IF xDeleteProcessFlag_St1St2 THEN
	xDeleteProcessFlag_St1St2:=FALSE;
	TProcess.T_Ctrle.xAbordProcess:=FALSE;
	TProcess.T_Ctrle.xStop:=FALSE;
END_IF;
END_ACTION
ACTION CtrlFunctionButton:
(* Bt Function Button *)
	xTmp:=	NOT(xChangePage)
			AND T_Visu.T_CtrleAction.xDone
			AND NOT(T_Visu.T_CtrleAction.xExecute);
	IF (wForceMaskFunctionPanel <> 0) THEN
		(* Wurde von einer Funktion überschrieben *)
		T_ConfigPage.wMaskFunctionPanel:=wForceMaskFunctionPanel;
		T_ConfigPage.wMaskProcFunctionPanel:=wForceMaskFunctionPanel;
		wMaskFunctionPanel:=wForceMaskFunctionPanel;
		wForceMaskFunctionPanel:=0;
	END_IF;
	FOR ii:=1 TO 12 DO
		IF (aiForceRTrigActionFunctionPanel[ii] <> 0) THEN
			(* Wurde von einer Funktion überschrieben *)
			T_ConfigPage.aiRTrigActionFunctionPanel:=aiForceRTrigActionFunctionPanel;
			EXIT;
		END_IF;
	END_FOR;
	aiForceRTrigActionFunctionPanel:=aiDelectRTrigActionFunctionPanel;
	RisingEdgeBtFunctionPanel(CLK:=	(T_ExchgParam.T_BtFunctionPanel.wActivBt
									AND wMaskFunctionPanel) <> 16#0);
	IF xTmp THEN
		(* check if more than one button is pressed-->if only one Button than start the procedure *)
		IF xFct_CheckSingleButtonActivation(wInputButton:=T_ExchgParam.T_BtFunctionPanel.wActivBt) THEN
		(* activ action of rising edge *)
			IF RisingEdgeBtFunctionPanel.Q AND NOT(xTriggerWait) THEN
				ii:=iFct_GetBitNumber(wInputButton:=T_ExchgParam.T_BtFunctionPanel.wActivBt);
				IF (T_ConfigPage.aiRTrigActionFunctionPanel[ii] <> 0) THEN
					T_Visu.T_CtrleAction.iFunction:=T_ConfigPage.aiRTrigActionFunctionPanel[ii];
					T_Visu.T_CtrleAction.xExecute:=TRUE;
				END_IF;
			END_IF;
		END_IF;
	END_IF
END_ACTION
ACTION CtrlPanelLeftButton:
(* Bt Panel left *)
	xTmp:=	NOT(xChangePage)
			AND T_Visu.T_CtrleAction.xDone
			AND NOT(T_Visu.T_CtrleAction.xExecute)
			AND NOT(T_StartUp.T_State.xBlockChangeMovementVisu)
			AND NOT(T_Visu.T_CtrleAction.xFunctionActive)
			AND (T_ExchgParam.T_Visu.T_Message.iState <> 401)
			AND ((T_ExchgParam.T_Visu.bMachineState AND 16#2) <> 16#2);
	xParameterButtonBlocked:=NOT(xTmp);
	RisingEdgeBtPanelLeft(CLK:=		(wActivBtLeft
									AND wMaskBtPanelLeft) <> 16#0);

	FallingEdgeBtPanelLeft(CLK:=		(wActivBtLeft
									AND wMaskBtPanelLeft) <> 16#0);
	IF RisingEdgeBtPanelLeft.Q THEN
		wActivBtPanelLeft:=wActivBtLeft;
	END_IF;
	IF xTmp THEN
		(* check if more than one button is pressed-->if only one Button than start the procedure *)
		IF xFct_CheckSingleButtonActivation(wInputButton:=wActivBtPanelLeft) THEN
		(* activ action of rising edge *)
			IF RisingEdgeBtPanelLeft.Q THEN
				ii:=iFct_GetBitNumber(wInputButton:=wActivBtPanelLeft);
				IF (T_ConfigPage.aiRTrigActionPanelLeft[ii] <> 0) THEN
					T_Visu.T_CtrleAction.iFunction:=T_ConfigPage.aiRTrigActionPanelLeft[ii];
					T_Visu.T_CtrleAction.xExecute:=TRUE;
				END_IF;
			END_IF;
		END_IF;
	END_IF

(* Aktivierungsanzeige für Maschinen Lampe *)
	IF TMachineLamp.T_CtrleCyl.T_Standard.xActivOn THEN
		T_ExchgParam.T_TouchScreenBtPanel.iStateSetupLamp:=1;
	ELSE
		T_ExchgParam.T_TouchScreenBtPanel.iStateSetupLamp:=0;
	END_IF;

(* Auswahl der Seiten über die Recht Sondertasten *)
T_ExchgParam.T_TouchScreenBtPanel.iStateButtonPage:=0;
CASE T_Visu.T_PlcParam.dwActualPage OF
(* NormalMode	Task 1 *)
gT_PageNumber.iAutoMode_Process:				T_ExchgParam.T_TouchScreenBtPanel.iStateButtonPage:=16#20;
gT_PageNumber.iAutoMode_ProcessValue1:			T_ExchgParam.T_TouchScreenBtPanel.iStateButtonPage:=16#40;		(* IGS *)
gT_PageNumber.iAutoMode_ProcessValue2:			T_ExchgParam.T_TouchScreenBtPanel.iStateButtonPage:=16#80;		(* IGS *)
gT_PageNumber.iAutoMode_PartQuality:				T_ExchgParam.T_TouchScreenBtPanel.iStateButtonPage:=16#100;		(* alt 80 *)
(* NormalMode	Task 4 *)
gT_PageNumber.iAutoMode_ToolChange:			T_ExchgParam.T_TouchScreenBtPanel.iStateButtonPage:=16#20;
gT_PageNumber.iAutoMode_UserLevel:				T_ExchgParam.T_TouchScreenBtPanel.iStateButtonPage:=16#40;
gT_PageNumber.iAutoMode_Language:				T_ExchgParam.T_TouchScreenBtPanel.iStateButtonPage:=16#80;
(* NormalMode	Task 5 *)
gT_PageNumber.iAutoMode_WPCounter:				T_ExchgParam.T_TouchScreenBtPanel.iStateButtonPage:=16#20;
gT_PageNumber.iAutoMode_LampTest:				T_ExchgParam.T_TouchScreenBtPanel.iStateButtonPage:=16#40;
gT_PageNumber.iAutoMode_SafetyCheck:			T_ExchgParam.T_TouchScreenBtPanel.iStateButtonPage:=16#80;
gT_PageNumber.iAutoMode_SysInfo:				T_ExchgParam.T_TouchScreenBtPanel.iStateButtonPage:=16#100;

(* SetupMode A	Task 1 *)
gT_PageNumber.iHandMode_Process:				T_ExchgParam.T_TouchScreenBtPanel.iStateButtonPage:=16#20;
gT_PageNumber.iHandMode_WorkParameter:		T_ExchgParam.T_TouchScreenBtPanel.iStateButtonPage:=16#40;
gT_PageNumber.iHandMode_RegulatorPara:			T_ExchgParam.T_TouchScreenBtPanel.iStateButtonPage:=16#80;
gT_PageNumber.iHandMode_OnlineChange:			T_ExchgParam.T_TouchScreenBtPanel.iStateButtonPage:=16#100;	(* alt 40 *)
gT_PageNumber.iHandMode_ConfigPosition:			T_ExchgParam.T_TouchScreenBtPanel.iStateButtonPage:=16#200;	(* alt 80 *)

(* SetupMode B	Task 5 *)
gT_PageNumber.iWorkStation_Setup1:				T_ExchgParam.T_TouchScreenBtPanel.iStateButtonPage:=16#20;
gT_PageNumber.iWorkStation_Setup2:				T_ExchgParam.T_TouchScreenBtPanel.iStateButtonPage:=16#40;
gT_PageNumber.iWorkStation_Setup3:				T_ExchgParam.T_TouchScreenBtPanel.iStateButtonPage:=16#80;
gT_PageNumber.iWorkStation_Setup4:				T_ExchgParam.T_TouchScreenBtPanel.iStateButtonPage:=16#100;
gT_PageNumber.iWorkStation_Setup5:				T_ExchgParam.T_TouchScreenBtPanel.iStateButtonPage:=16#200;
END_CASE;
END_ACTION
ACTION CtrlPanelRightButton:
(* Bt Panel right *)
	xTmp:=	NOT(xChangePage)
			AND T_Visu.T_CtrleAction.xDone
			AND NOT(T_Visu.T_CtrleAction.xExecute);
	IF (wForceMaskBtPanelRight <> 0) THEN
		(* Wurde von einer Funktion überschrieben *)
		T_ConfigPage.wMaskBtPanelRight:=wForceMaskBtPanelRight;
		T_ConfigPage.wMaskProcBtPanelRight:=wForceMaskBtPanelRight;
		wMaskBtPanelRight:=wForceMaskBtPanelRight;
		wForceMaskBtPanelRight:=0;
	END_IF;
	FOR ii:=1 TO 5 DO
		IF (aiForceRTrigActionPanelRight[ii] <> 0) THEN
			(* Wurde von einer Funktion überschrieben *)
			T_ConfigPage.aiRTrigActionPanelRight:=aiForceRTrigActionPanelRight;
			EXIT;
		END_IF;
	END_FOR;
	aiForceRTrigActionPanelRight:=aiDeleteRTrigActionPanelRight;

	xActive_Joystick:=			IxJoystick_X_Plus OR IxJoystick_X_Minus OR IxJoystick_Y_Plus OR IxJoystick_Y_Minus;
	xActive_EnableSwitch:=		IxEnablingSwitchPlusButton OR IxEnablingSwitchMinusButton;

	IF (wActivBtRight = 0) AND NOT(xActive_EnableSwitch) THEN
		(* Achsenbewegung mit dem Joystick *)
		IF IxJoystick_Y_Plus AND NOT(IxJoystick_Y_Minus) AND gxEnable_Joystick_Axis_Z THEN
			wActivBtRight:=16#40;
			T_ConfigPage.aiRTrigActionPanelRight[2]:=216;
			wMaskBtPanelRight:=wActivBtRight;
		END_IF;
		IF NOT(IxJoystick_Y_Plus) AND IxJoystick_Y_Minus AND gxEnable_Joystick_Axis_Z THEN
			wActivBtRight:=16#20;
			T_ConfigPage.aiRTrigActionPanelRight[1]:=217;
			wMaskBtPanelRight:=wActivBtRight;
		END_IF;
		IF (IxJoystick_Y_Plus OR IxJoystick_Y_Minus) AND NOT(gxEnable_Joystick_Axis_Z) AND (T_ExchgParam.T_Visu.T_Message.iState <> 401) THEN
			T_ExchgParam.T_Visu.T_Message.iState:=306;	(* Warnung: Z Achse darf auf dieser Seite nicht verfahren werden ! *)
		END_IF;
	END_IF;

	IF (T_Visu.T_PlcParam.dwActualPage = gT_PageNumber.iWorkStation_Axis1) THEN
		gxReleaseEnableSwitch:=TRUE;
	ELSE
		gxReleaseEnableSwitch:=FALSE;
	END_IF;

	IF gxReleaseEnableSwitch AND (wActivBtRight = 0) AND NOT(xActive_Joystick) AND gT_SafetyStatus.xSecurityDoorOpen THEN
		(* Achsenbewegung mit dem Zustimmschalter *)
		IF IxEnablingSwitchPlusButton AND NOT(IxEnablingSwitchMinusButton) THEN
			wActivBtRight:=16#40;
			T_ConfigPage.aiRTrigActionPanelRight[2]:=216;
		END_IF;
		IF NOT(IxEnablingSwitchPlusButton) AND IxEnablingSwitchMinusButton THEN
			wActivBtRight:=16#20;
			T_ConfigPage.aiRTrigActionPanelRight[1]:=217;
		END_IF;
	END_IF;

	RisingEdgeBtPanelRight(CLK:=		(wActivBtRight
									AND wMaskBtPanelRight) <> 16#0);
	FallingEdgeBtPanelRight(CLK:=		(wActivBtRight
									AND wMaskBtPanelRight) <> 16#0);
	IF xTmp THEN
		(* check if more than one button is pressed-->if only one Button than start the procedure *)
		IF xFct_CheckSingleButtonActivation(wInputButton:=wActivBtRight) THEN
		(* activ action of rising edge *)
			IF RisingEdgeBtPanelRight.Q THEN
				ii:=iFct_GetBitNumber(wInputButton:=wActivBtRight) - 5;
				wActivBtPanelRight:=INT_TO_WORD(ii);
				IF (T_ConfigPage.aiRTrigActionPanelRight[ii] <> 0) THEN
					T_Visu.T_CtrleAction.iFunction:=T_ConfigPage.aiRTrigActionPanelRight[ii];
					T_Visu.T_CtrleAction.xExecute:=TRUE;
					xJogModeActive:=xFct_GetJogMode(iFunction:=T_Visu.T_CtrleAction.iFunction);
					wSaveBtPanelRight:=wActivBtRight;
				END_IF;
			END_IF;
		END_IF;
		(* activ action of failling edge *)
		IF FallingEdgeBtPanelRight.Q THEN
			ii:=WORD_TO_INT(wActivBtPanelRight);
			IF (T_ConfigPage.aiFTrigActionPanelRight[ii] <> 0) THEN
				T_Visu.T_CtrleAction.iFunction:=T_ConfigPage.aiFTrigActionPanelRight[ii];
				T_Visu.T_CtrleAction.xExecute:=TRUE;
			END_IF;
		END_IF;
	END_IF

(* Überprüfe wenn Jog Betrieb gestartet ist, dass wenn die Taste nicht mehr gedrückt ist, dass die Achse auch gestoppt wird-->Falls nicht, dann muss es explizit gestoppt werden *)
	IF xJogModeActive OR xTmpJogModeActive THEN
		CASE iStepJogModeActive OF
		1:	IF NOT(xInitJogVelocity) THEN
				xInitJogVelocity:=TRUE;
				lrJogVelocity:=T_ExchgParam.T_TeachIn.arTeachSelVel[ptrTCommonAxisActive^.T_Config_Gen.iTyp];
			END_IF;
			xJogModeActive:=FALSE;
			xTmpJogModeActive:=TRUE;
			IF ((wSaveBtPanelRight AND wActivBtRight) = 16#0) THEN
				(* Taste wurde losgelassen *)
				iStepJogModeActive:=iStepJogModeActive + 1;
				RETURN;
			END_IF;
			IF T_ExchgParam.T_TeachIn.xJogInc_Common_Setup_Axis AND (lrJogVelocity <> T_ExchgParam.T_TeachIn.arTeachSelVel[ptrTCommonAxisActive^.T_Config_Gen.iTyp]) THEN
				lrJogVelocity:=T_ExchgParam.T_TeachIn.arTeachSelVel[ptrTCommonAxisActive^.T_Config_Gen.iTyp];
				(* Jog-Betrieb ist ausgewählt-->Geschwindigkeit in Abhängigkeit des Poti einstellen *)
				IF NOT(ptrTCommonAxisActive^.T_CtrleSingle.xExecute) AND ptrTCommonAxisActive^.T_CtrleSingle.xDone AND
				     NOT(ptrTCommonAxisActive^.T_CtrleSingle.xErr) AND NOT(ptrTCommonAxisActive^.T_CtrleSingle.xNotMoving) THEN
					ptrTCommonAxisActive^.T_CtrleSingle.iFunction:=12;
					gxSetSpeedInMovement:=TRUE;
					IF ptrTCommonAxisActive^.T_CtrleSingle.xMovingForward THEN
						ptrTCommonAxisActive^.T_CtrleSingle.lrVelocity:=T_ExchgParam.T_TeachIn.arTeachSelVel[ptrTCommonAxisActive^.T_Config_Gen.iTyp];
					ELSE
						ptrTCommonAxisActive^.T_CtrleSingle.lrVelocity:=T_ExchgParam.T_TeachIn.arTeachSelVel[ptrTCommonAxisActive^.T_Config_Gen.iTyp]*-1.0;
					END_IF;
					ptrTCommonAxisActive^.T_CtrleSingle.xExecute:=TRUE;
				END_IF;
			END_IF;
		2:	IF ((ptrTCommonAxisActive^.T_CtrleSingle.iFunction = 6) OR (ptrTCommonAxisActive^.T_CtrleSingle.iFunction = 12)) AND NOT(ptrTCommonAxisActive^.T_CtrleSingle.xNotMoving) AND NOT(xJogModeActive) THEN
				T_Visu.T_CtrleAction.iFunction:=202;	(* Stoppen aller Achse *)
				T_Visu.T_CtrleAction.xExecute:=TRUE;
				xTmpJogModeActive:=FALSE;
				iStepJogModeActive:=1;
			END_IF
			IF (ptrTCommonAxisActive^.T_CtrleSingle.iFunction <> 6) AND (ptrTCommonAxisActive^.T_CtrleSingle.iFunction <> 12) AND NOT(xJogModeActive) THEN
				(* Es wurde ein Inkrementfahrt ausgelöst und daher muss es nicht explizit gestoppt werden *)
				xTmpJogModeActive:=FALSE;
				iStepJogModeActive:=1;
			END_IF;
			IF xJogModeActive THEN
				iStepJogModeActive:=1;	(* Jog wurde vor dem beenden wieder gestartet, daher muss es wieder überprüft werden *)
				xInitJogVelocity:=FALSE;
			END_IF;
		END_CASE;
	ELSE
		iStepJogModeActive:=1;
		xInitJogVelocity:=FALSE;
	END_IF;

(* Verwaltung der Freigabe für den Joystick *)
	IF NOT(T_StartUp.T_State.xCompleted) THEN
		(* Solange die Maschine nicht aufgestartet ist, ist die manuelle Achsenbewegung nicht erlaubt *)
		xResetEnableJoystickAxisZ:=TRUE;
		xSetEnableJoystickAxisZ:=FALSE;
	ELSIF NOT(gT_SafetyStatus.xSetupOperateModeActive) THEN
		(* Im NormalBetrieb ist die manuelle Achsenbewegung nicht erlaubt *)
		xResetEnableJoystickAxisZ:=TRUE;
		xSetEnableJoystickAxisZ:=FALSE;
	ELSIF gT_SafetyStatus.xSetupOperateModeActive AND (gT_SafetyStatus.iSetupMode = 1) THEN
		(* Im EinrichtBetrieb A ist die manuelle Achsenbewegung nur unter dem Task HandBetrieb erlaubt *)
		xResetEnableJoystickAxisZ:=TRUE;
		xSetEnableJoystickAxisZ:=FALSE;
		IF TStation_Work_St1.TControl.xEnable AND TStation_Work_St1.TControl.xRdy AND TStation_Work_St1.TControl.xDone AND NOT(TStation_Work_St1.TControl.xError) THEN
			IF (T_Visu.T_PlcParam.dwActualPage = gT_PageNumber.iHandMode_Process)
			OR (T_Visu.T_PlcParam.dwActualPage = gT_PageNumber.iHandMode_WorkParameter) OR (T_Visu.T_PlcParam.dwActualPage = gT_PageNumber.iHandMode_RegulatorPara)
			OR (T_Visu.T_PlcParam.dwActualPage = gT_PageNumber.iHandMode_OnlineChange) OR (T_Visu.T_PlcParam.dwActualPage = gT_PageNumber.iHandMode_ConfigPosition) THEN
				xResetEnableJoystickAxisZ:=FALSE;
				xSetEnableJoystickAxisZ:=TRUE;
			END_IF;
		END_IF;
	ELSIF gT_SafetyStatus.xSetupOperateModeActive AND (gT_SafetyStatus.iSetupMode = 2) THEN
		(* Im EinrichtBetrieb B ist die manuelle Achsenbewegung erlaubt sofern nicht eine Funktion am ausführen ist *)
		IF NOT(TStation_Work_St1.TControl.xEnable) OR NOT(TStation_Work_St1.TControl.xRdy) OR NOT(TStation_Work_St1.TControl.xDone) OR  TStation_Work_St1.TControl.xError THEN
			xResetEnableJoystickAxisZ:=TRUE;
			xSetEnableJoystickAxisZ:=FALSE;
		ELSE
			xResetEnableJoystickAxisZ:=FALSE;
			xSetEnableJoystickAxisZ:=TRUE;
		END_IF;
		IF xTmpStationSetupAxisZFunction AND (T_ExchgParam.T_StationCommon.iZAxisFirstSetup_ShowObjectNr = 3) THEN
			xResetEnableJoystickAxisZ:=FALSE;
			xSetEnableJoystickAxisZ:=TRUE;
		END_IF;
		IF xTmpStationSetupAxisZFunction AND (T_ExchgParam.T_StationCommon.iZAxisFirstSetup_ShowObjectNr <> 3) THEN
			xResetEnableJoystickAxisZ:=TRUE;
			xSetEnableJoystickAxisZ:=FALSE;
		END_IF;
		IF xTmpStationSetupAxisZFunctionToolGuide AND (T_ExchgParam.T_StationCommon.iZAxisGuideTube_ShowObjectNr = 6) THEN
			xResetEnableJoystickAxisZ:=FALSE;
			xSetEnableJoystickAxisZ:=TRUE;
		END_IF;
		IF xTmpStationSetupAxisZFunctionToolGuide AND (T_ExchgParam.T_StationCommon.iZAxisGuideTube_ShowObjectNr <> 6) THEN
			xResetEnableJoystickAxisZ:=TRUE;
			xSetEnableJoystickAxisZ:=FALSE;
		END_IF;
	ELSE
		(* Alles restliche ist nicht erlaubt *)
		xResetEnableJoystickAxisZ:=TRUE;
		xSetEnableJoystickAxisZ:=FALSE;
	END_IF;

	IF xSetEnableJoystickAxisZ THEN
		gxEnable_Joystick_Axis_Z:=TRUE;
	END_IF;
	IF xResetEnableJoystickAxisZ OR NOT(T_StartUp.T_Ctrle.xDone) THEN
		gxEnable_Joystick_Axis_Z:=FALSE;
	END_IF;
END_ACTION
ACTION CtrlParaListButton:
IF NOT(xSecurityKey) THEN
	iStationActive:=0;
ELSE
	iStationActive:=iSetupMode;
END_IF;
(* Bt Parameter List Button *)
	xTmp:=	NOT(xChangePage)
			AND T_Visu.T_CtrleAction.xDone
			AND NOT(T_Visu.T_CtrleAction.xExecute);
	RisingEdgeBtParameterList(CLK:=	(T_ExchgParam.T_BtParameterList.wActivBt<>0));
	IF xTmp THEN
		(* check if more than one button is pressed-->if only one Button than start the procedure *)
		IF xFct_CheckSingleButtonActivation(wInputButton:=T_ExchgParam.T_BtParameterList.wActivBt) THEN
		(* activ action of rising edge *)
			IF RisingEdgeBtParameterList.Q THEN
				ii:=iFct_GetBitNumber(wInputButton:=T_ExchgParam.T_BtParameterList.wActivBt);
				jj:=iFct_GetBitNumber(wInputButton:=awSaveStateTaskBar[iStationActive]);
(*				aiTempActiveParaListState[iStationActive,jj]:=ii;*)
				(* Da diese Software keine Parameterlisten bezogen auf Task hat, sind alle gleichgestellt *)
				aiTempActiveParaListState[iStationActive,1]:=ii;
				aiTempActiveParaListState[iStationActive,2]:=ii;
				aiTempActiveParaListState[iStationActive,3]:=ii;
				aiTempActiveParaListState[iStationActive,4]:=ii;
				aiTempActiveParaListState[iStationActive,5]:=ii;
				aiTempActiveParaListState[iStationActive,6]:=ii;
				xUpdateStationParameter:=TRUE;
			END_IF;
		END_IF;
		T_ExchgParam.T_BtParameterList.wActivBt:=0;
	ELSE
		T_ExchgParam.T_BtParameterList.wActivBt:=0;
	END_IF

FBGetParameterList(	xNormalModeActive:= NOT(xSecurityKey),
					iSetupMode:= iSetupMode,
					wActiveTaskBar:= awSaveStateTaskBar[iStationActive],
					aiTempActiveParaListState:= aiTempActiveParaListState,
					iActLevel:=T_ExchgParam.T_Visu.T_Level.iActLevel);
T_ExchgParam.T_BtParameterList.iEditParam:=FBGetParameterList.iParameterList;
T_ExchgParam.T_BtParameterList.wNotMasktext:=FBGetParameterList.wNotMasktext;
T_ExchgParam.T_BtParameterList.wState:=FBGetParameterList.wState;
T_ExchgParam.T_BtParameterList.aiSelectText:=FBGetParameterList.aiSelectText;
T_ExchgParam.T_BtParameterList.bParameterListEditable:=FBGetParameterList.bParameterListEditable;
T_ExchgParam.T_BtParameterList.bMessageParameter:=FBGetParameterList.bMessageParameter;
END_ACTION
ACTION CtrlPreWarning:
(* Ausgabe der Vorwarnungsmeldungen *)
IF T_ExchgParam.T_SafetyCtrl.xReadNextPreWarningMessage THEN
	T_ExchgParam.T_SafetyCtrl.xReadNextPreWarningMessage:=FALSE;
	IF gT_PreWarning.xPreWarningActive THEN
		iMessageSelected:=iMessageSelected + 1;
		IF (iMessageSelected > gT_PreWarning.iNumberOfMessage) THEN
			iMessageSelected:=gT_PreWarning.iNumberOfMessage;
		END_IF;
	END_IF;
END_IF;
IF T_ExchgParam.T_SafetyCtrl.xReadPreviousPreWarningMessage THEN
	T_ExchgParam.T_SafetyCtrl.xReadPreviousPreWarningMessage:=FALSE;
	IF gT_PreWarning.xPreWarningActive THEN
		iMessageSelected:=iMessageSelected - 1;
		IF (iMessageSelected < 1) THEN
			iMessageSelected:=1;
		END_IF;
	END_IF;
END_IF;
IF (iMessageSelected > gT_PreWarning.iNumberOfMessage) THEN
	iMessageSelected:=gT_PreWarning.iNumberOfMessage;
END_IF;
IF (iMessageSelected = 0) AND (gT_PreWarning.iNumberOfMessage > 0) THEN
	iMessageSelected:=1;
END_IF;
IF NOT(gT_PreWarning.xPreWarningActive) THEN
	T_ExchgParam.T_SafetyCtrl.sDynMsgPreWarningLine1Engl:=gT_PreWarning.asEmptyMessageEngl[1];
	T_ExchgParam.T_SafetyCtrl.sDynMsgPreWarningLine2Engl:=gT_PreWarning.asEmptyMessageEngl[2];
	T_ExchgParam.T_SafetyCtrl.sDynMsgPreWarningLine3Engl:=gT_PreWarning.asEmptyMessageEngl[3];
	T_ExchgParam.T_SafetyCtrl.sDynMsgPreWarningLine4Engl:=gT_PreWarning.asEmptyMessageEngl[4];
	T_ExchgParam.T_SafetyCtrl.sDynMsgPreWarningLine5Engl:=gT_PreWarning.asEmptyMessageEngl[5];
	T_ExchgParam.T_SafetyCtrl.sDynMsgPreWarningLine1Ger:=gT_PreWarning.asEmptyMessageGer[1];
	T_ExchgParam.T_SafetyCtrl.sDynMsgPreWarningLine2Ger:=gT_PreWarning.asEmptyMessageGer[2];
	T_ExchgParam.T_SafetyCtrl.sDynMsgPreWarningLine3Ger:=gT_PreWarning.asEmptyMessageGer[3];
	T_ExchgParam.T_SafetyCtrl.sDynMsgPreWarningLine4Ger:=gT_PreWarning.asEmptyMessageGer[4];
	T_ExchgParam.T_SafetyCtrl.sDynMsgPreWarningLine5Ger:=gT_PreWarning.asEmptyMessageGer[5];
ELSE
	sWrapTextEngl:='Message ';
	sWrapTextEngl:=CONCAT(sWrapTextEngl, INT_TO_STRING(iMessageSelected));
	sWrapTextEngl:=CONCAT(sWrapTextEngl, ' of ');
	sWrapTextEngl:=CONCAT(sWrapTextEngl, INT_TO_STRING(gT_PreWarning.iNumberOfMessage));
	T_ExchgParam.T_SafetyCtrl.sDynMsgPreWarningLine1Engl:=sWrapTextEngl;
	T_ExchgParam.T_SafetyCtrl.sDynMsgPreWarningLine2Engl:=gT_PreWarning.asMessageBufferEngl[iMessageSelected,2];
	T_ExchgParam.T_SafetyCtrl.sDynMsgPreWarningLine3Engl:=gT_PreWarning.asMessageBufferEngl[iMessageSelected,3];
	T_ExchgParam.T_SafetyCtrl.sDynMsgPreWarningLine4Engl:=gT_PreWarning.asMessageBufferEngl[iMessageSelected,4];
	T_ExchgParam.T_SafetyCtrl.sDynMsgPreWarningLine5Engl:=gT_PreWarning.asMessageBufferEngl[iMessageSelected,5];
	sWrapTextGer:='Meldung ';
	sWrapTextGer:=CONCAT(sWrapTextGer, INT_TO_STRING(iMessageSelected));
	sWrapTextGer:=CONCAT(sWrapTextGer, ' von ');
	sWrapTextGer:=CONCAT(sWrapTextGer, INT_TO_STRING(gT_PreWarning.iNumberOfMessage));
	T_ExchgParam.T_SafetyCtrl.sDynMsgPreWarningLine1Ger:=sWrapTextGer;
	T_ExchgParam.T_SafetyCtrl.sDynMsgPreWarningLine2Ger:=gT_PreWarning.asMessageBufferGer[iMessageSelected,2];
	T_ExchgParam.T_SafetyCtrl.sDynMsgPreWarningLine3Ger:=gT_PreWarning.asMessageBufferGer[iMessageSelected,3];
	T_ExchgParam.T_SafetyCtrl.sDynMsgPreWarningLine4Ger:=gT_PreWarning.asMessageBufferGer[iMessageSelected,4];
	T_ExchgParam.T_SafetyCtrl.sDynMsgPreWarningLine5Ger:=gT_PreWarning.asMessageBufferGer[iMessageSelected,5];
END_IF;
IF T_ExchgParam.T_SafetyCtrl.xResetMsgPreWarning THEN
	T_ExchgParam.T_SafetyCtrl.xResetMsgPreWarning:=FALSE;
	IF gT_PreWarning.xPreWarningActive AND (iMessageSelected <> 0) THEN
		giDeleteMessageNumber:=giDeleteMessageNumber + 1;
		gT_PreWarning.aiDeleteMessage[giDeleteMessageNumber]:=gT_PreWarning.aiMessageNrBuffer[iMessageSelected];
	END_IF;
END_IF;
IF T_ExchgParam.T_SafetyCtrl.xConfirmMsgPreWarning THEN
	T_ExchgParam.T_SafetyCtrl.xConfirmMsgPreWarning:=FALSE;
	T_ExchgParam.T_SafetyCtrl.bStateMessagePreWarning:=0;
END_IF;
IF (T_ExchgParam.T_SafetyCtrl.bStateMessageError <> 0) OR (T_ExchgParam.T_SafetyCtrl.bStateMessageInfo <> 0) OR (T_ExchgParam.T_SafetyCtrl.bStateMessageWarning <> 0) THEN
	T_ExchgParam.T_SafetyCtrl.xConfirmMsgPreWarning:=FALSE;
	T_ExchgParam.T_SafetyCtrl.bStateMessagePreWarning:=0;
END_IF;
END_ACTION
ACTION CtrlProcessFunction:
(* Manage process execution *)
	(* ...done *)
	RisingEdgeProcessDone(CLK:=T_Visu.T_CtrleProcess.xDone);
	IF RisingEdgeProcessDone.Q THEN
		;
	END_IF
	(* ...error *)
	RisingEdgeProcessError(CLK:=T_Visu.T_CtrleProcess.xErr);
	IF RisingEdgeProcessError.Q THEN
		(* Init. variable *)
		T_Visu.T_CtrleProcess.xExecute:=FALSE;
		T_Visu.T_CtrleProcess.xDone:=TRUE;
		T_Visu.T_CtrleProcess.xErr:=FALSE;
		T_Visu.T_CtrleProcess.udiErrorID:=0;
		iStepProcess:=1;
		xStepProcessDone:=FALSE;
	END_IF
	(* ...reset *)
	RisingEdgeReseTProcess(CLK:=T_Visu.T_CtrleProcess.xReset);
	IF RisingEdgeReseTProcess.Q THEN
		(* Init. variable *)
		T_Visu.T_CtrleProcess.xExecute:=FALSE;
		T_Visu.T_CtrleProcess.xDone:=TRUE;
		T_Visu.T_CtrleProcess.xErr:=FALSE;
		T_Visu.T_CtrleProcess.udiErrorID:=0;
		iStepProcess:=1;
		xStepProcessDone:=FALSE;
		(* Release process *)
		T_Visu.T_CtrleProcess.xReset:=FALSE;
		xProcessMachine:=FALSE;
		xProcessStation:=FALSE;
	END_IF
	RisingEdgeExecuteProcess(CLK:=T_Visu.T_CtrleProcess.xExecute);
	IF RisingEdgeExecuteProcess.Q THEN
		(* Release execution *)
		T_Visu.T_CtrleProcess.xExecute:=FALSE;
		CASE T_Visu.T_CtrleProcess.iFunction OF
		(* Process machine *)
		1:	xProcessMachine:=TRUE;
		(* Process station mit WstkTeller *)
		2:	xProcessStation:=TRUE;
		(* process not implemented *)
		ELSE	T_Visu.T_CtrleProcess.xDone:=FALSE;
				T_Visu.T_CtrleProcess.xErr:=TRUE;
				T_Visu.T_CtrleProcess.udiErrorID:=16#E000;
				(* exit FB *)
				RETURN;
		END_CASE
		(* Init. variable *)
		T_Visu.T_CtrleProcess.xDone:=FALSE;
		T_Visu.T_CtrleProcess.xErr:=FALSE;
		T_Visu.T_CtrleProcess.udiErrorID:=0;
		iStepProcess:=1;
		xStepProcessDone:=FALSE;
		(* exit FB *)
		RETURN;
	END_IF

(* Prozesse die im Einrichtbetrieb ausgelöst werden mit dem WstkTeller *)
	IF xProcessStation THEN
		IF NOT(TProcess.T_Ctrle.xExecute)  AND TProcess.T_Ctrle.xError AND TProcess.T_Ctrle.xErrorReady THEN
			iStepProcess:=90;
		END_IF;
		CASE iStepProcess OF
		1:	TProcess.T_Ctrle.xExecute:=TRUE;	(* Starten des Prozesses *)
			iStepProcess:=90;
		(* Abwarten auf das Prozessende *)
		90:	IF NOT(TProcess.T_Ctrle.xExecute)  AND (TProcess.T_Ctrle.xDone OR TProcess.T_Ctrle.xError) THEN
				T_StartUp.T_State.xBlockChangeMovementVisu:=FALSE;
				xProcessStation:=FALSE;
				T_Visu.T_CtrleProcess.xDone:=TRUE;
				T_Visu.T_CtrleProcess.xErr:=FALSE;
				T_Visu.T_CtrleProcess.udiErrorID:=0;
			END_IF;
			IF (T_ExchgParam.byOverride = 0) THEN
				T_ExchgParam.T_Visu.T_Message.iState:=330;	(* Override ist auf 0% gesetzt-->Keine Achsenbewegung ! *)
			ELSE
				IF (T_ExchgParam.T_Visu.T_Message.iState = 330) THEN
					T_ExchgParam.T_Visu.T_Message.iState:=0;
				END_IF;
			END_IF;
		END_CASE;
	END_IF;

(* Prozesse die im Automat ausgelöst werden *)
	IF xProcessMachine THEN
		CASE iStepProcess OF
		(* Überprüfe zuerst den WzWechsel der Bearbeitungsstationen *)
		1:	xProcessEnded:=FALSE;
			IF (TProcess.T_Ctrle.iFunctNr = 2) THEN
				(* Gilt nur für den Automat *)
				T_ExchgParam.T_Visu.T_Message.iState:=0;
				T_ExchgParam.T_StationCommon.T_ToolCounter_St1.diToolCycleCounter:=T_NovRam.T_Parameter.T_StationWork[gciStationSt1].T_ToolCounter.diToolCycleCounter;
				T_ExchgParam.T_StationCommon.T_ToolCounter_St1.diMaxNumberToolCycle:=T_NovRam.T_Parameter.T_StationWork[gciStationSt1].T_ToolCounter.diMaxNumberToolCycle;
				xTmp:=	((T_NovRam.T_Parameter.T_StationWork[gciStationSt1].T_ToolCounter.diMaxNumberToolCycle <> 0) AND
						(T_NovRam.T_Parameter.T_StationWork[gciStationSt1].T_ToolCounter.diToolCycleCounter >= T_NovRam.T_Parameter.T_StationWork[gciStationSt1].T_ToolCounter.diMaxNumberToolCycle));
				IF xTmp THEN
					T_ExchgParam.T_SafetyCtrl.bStateMessageRequest:=1;
					T_ExchgParam.T_SafetyCtrl.bStateMessagePreWarning:=0;
					T_StartUp.T_State.xBlockChangeMovementVisu:=TRUE;
					iStepProcess:=iStepProcess + 1;
				ELSE
					iStepProcess:=4;	(* Überprüfen des Namen für die Prozessanalyse *)
				END_IF;
			ELSE
					iStepProcess:=19;	(* Prozess kann gestartet werden *)
			END_IF;
			xProcessAbordet:=FALSE;
		(* Aufforderung an Operator für Eingabe ob WzWechsel stattgefunden hat oder nicht *)
		2:	IF T_ExchgParam.T_SafetyCtrl.xConfirmMsgRequest THEN
				T_ExchgParam.T_SafetyCtrl.xConfirmMsgRequest:=FALSE;
				T_ExchgParam.T_SafetyCtrl.bStateMessageRequest:=0;
				IF (T_ExchgParam.T_SafetyCtrl.bState_Select_St1 = 1) THEN
					T_NovRam.T_Parameter.T_StationWork[gciStationSt1].T_ToolCounter.diToolCycleCounter:=0;
					T_ExchgParam.T_StationCommon.T_ToolCounter_St1.diToolCycleCounter:=0;
				END_IF;
				TONWaitReadyStartButton(IN:=FALSE);
				T_ExchgParam.T_Visu.T_Message.iState:=101;	(* Aufforderung: Bitte StartTaste drücken um Prozess zu starten *)
				iStepProcess:=iStepProcess + 1;
			END_IF;
		(* Auffordern erneut die StartTaste zu drücken *)
		3:	T_CtrleBtStartStop.xForceSetStartButton:=TONWaitReadyStartButton.Q;
			T_CtrleBtStartStop.xForceSetStopButton:=TONWaitReadyStartButton.Q;
			T_ExchgParam.T_Visu.T_Message.iState:=101;	(* Aufforderung: Bitte StartTaste drücken um Prozess zu starten *)
			IF xStartButton THEN
				TONWaitReadyStartButton(IN:=FALSE);
				T_ExchgParam.T_Visu.T_Message.iState:=0;		(* Meldung zurücksetzen *)
				T_StartUp.T_State.xBlockChangeMovementVisu:=FALSE;
				iStepProcess:=4;
			END_IF;
			IF xStopButton THEN
				TONWaitReadyStartButton(IN:=FALSE);
				T_ExchgParam.T_Visu.T_Message.iState:=0;		(* Meldung zurücksetzen *)
				T_ExchgParam.T_Visu.T_Message.iState:=0;
				xProcessMachine:=FALSE;
				T_Visu.T_CtrleProcess.xDone:=TRUE;
				T_Visu.T_CtrleProcess.xErr:=FALSE;
				T_Visu.T_CtrleProcess.udiErrorID:=0;
				T_StartUp.T_State.xBlockChangeMovementVisu:=FALSE;
			END_IF;
		(* Überprüfe ob der Name für die Prozessanalyse eingegeben werden muss *)
		4:	IF (T_NovRam.T_Parameter.T_PartAnalysis[gciStationSt1].sStartOfProcess = '') THEN
				TStation_Work_St1.THWWorkStation.TCtrlWork.xWP_Analyse_StartAutomat:=TRUE;			(* Gilt für die Aufzeichnungsdatei, um festzulegen wann der Automat für die jeweilige Datei gestartet wurde *)
			END_IF;
			iStepProcess:=19;
		(* Sicherheitstüren Zuhaltung aktivieren *)
		19:	T_ExchgParam.T_SafetyCtrl.xCloseSecurityDoorMachine:=TRUE;
			iStepProcess:=20;
		20:	IF NOT(T_ExchgParam.T_SafetyCtrl.xCloseSecurityDoorMachine) THEN
				iStepProcess:=30;
			END_IF;
		(* Prozess starten *)
		30:	TProcess.T_Ctrle.xExecute:=TRUE;	(* Starten des Prozesses *)
			iStepProcess:=90;
		90:	IF NOT(TProcess.T_Ctrle.xExecute)  AND TProcess.T_Ctrle.xDone THEN
				xProcessEnded:=TRUE;
				IF NOT(xProcessAbordet) THEN
					IF (TProcess.T_Ctrle.iFunctNr = 1) THEN
						T_StartUp.T_Ctrle.iMsgNumber:=3;	(* Die Maschine wurde Referenziert/Grundstellung! Bestätigen Sie die Meldung und die Zuhaltung der MaschinenTüre wird deaktiviert! *)
						T_StartUp.T_Ctrle.iFunction:=11;
						T_StartUp.T_Ctrle.xExecute:=TRUE;
					ELSIF (TProcess.T_Ctrle.iFunctNr = 2) THEN
						T_StartUp.T_Ctrle.iMsgNumber:=10;	(* Das Leerfahren im Automat ist beendet! Bestätigen Sie die Meldung und die Zuhaltung der MaschinenTüre wird deaktiviert! *)
						T_StartUp.T_Ctrle.iFunction:=11;
						T_StartUp.T_Ctrle.xExecute:=TRUE;
					END_IF;
				ELSE
					xProcessAbordet:=FALSE;
					T_StartUp.T_Ctrle.iMsgNumber:=10;	(* Prozess wurde abgebrochen! Bestätigen Sie die Meldung und die Zuhaltung der MaschinenTüre wird deaktiviert! *)
					T_StartUp.T_Ctrle.iFunction:=12;
					T_StartUp.T_Ctrle.xExecute:=TRUE;
				END_IF;
				T_StartUp.T_Ctrle.xUnlockSecurityDoor:=TRUE;	(* Auffordern Sicherheitstüren zu öffnen, nachdem die Meldung vom Operator Quittiert wurde *)
				xProcessMachine:=FALSE;
				T_Visu.T_CtrleProcess.xDone:=TRUE;
				T_Visu.T_CtrleProcess.xErr:=FALSE;
				T_Visu.T_CtrleProcess.udiErrorID:=0;
				T_ExchgParam.T_StationCommon.xBlockSelectAutoMode:=FALSE;
			END_IF;
			IF NOT(TProcess.T_Ctrle.xExecute)  AND TProcess.T_Ctrle.xError AND TProcess.T_Ctrle.xErrorReady THEN
				xProcessEnded:=TRUE;
				IF (TProcess.T_Ctrle.iFunctNr = 1) THEN
					T_StartUp.T_Ctrle.iMsgNumber:=58;	(* Während der Maschinen Ref./Grundstellung ist ein Fehler/Error aufgetreten! Bestätigen Sie die Meldung und Überprüfen Sie den entsprechenden Fehler/Error *)
				ELSIF (TProcess.T_Ctrle.iFunctNr = 2) THEN
					T_StartUp.T_Ctrle.iMsgNumber:=55;	(* Während des Automat ist ein Fehler/Error aufgetreten! Bestätigen Sie die Meldung und Überprüfen Sie den entsprechenden Fehler/Error *)
				END_IF;
				T_StartUp.T_Ctrle.iFunction:=10;
				T_StartUp.T_Ctrle.xUnlockSecurityDoor:=TRUE;	(* Auffordern Sicherheitstüren zu öffnen, nachdem die Meldung vom Operator Quittiert wurde *)
				T_StartUp.T_Ctrle.xExecute:=TRUE;
				xProcessMachine:=FALSE;
				T_Visu.T_CtrleProcess.xDone:=TRUE;
				T_Visu.T_CtrleProcess.xErr:=FALSE;
				T_Visu.T_CtrleProcess.udiErrorID:=0;
				T_ExchgParam.T_StationCommon.xBlockSelectAutoMode:=FALSE;
			END_IF;
			IF (T_ExchgParam.byOverride = 0) THEN
				T_ExchgParam.T_Visu.T_Message.iState:=330;	(* Override ist auf 0% gesetzt-->Keine Achsenbewegung ! *)
			ELSE
				IF (T_ExchgParam.T_Visu.T_Message.iState = 330) THEN
					T_ExchgParam.T_Visu.T_Message.iState:=0;
				END_IF;
			END_IF;
		END_CASE;
	END_IF;

	IF (T_StartUp.T_Ctrle.iMsgNumber = 10) AND (T_StartUp.T_Ctrle.iFunction = 11) AND NOT(T_StartUp.T_Ctrle.xDone) AND T_StartUp.T_State.xCompleted AND NOT(gT_SafetyStatus.xSetupOperateModeActive) AND NOT(T_ExchgParam.T_SafetyCtrl.xConfirmMsgInfo) THEN
		TONWaitSwitchOffMessage(IN:=TRUE,PT:=T#3s);
		IF TONWaitSwitchOffMessage.Q THEN
			T_ExchgParam.T_SafetyCtrl.xConfirmMsgInfo:=TRUE;
			TONWaitSwitchOffMessage(IN:=FALSE);
		END_IF;
	ELSE
		TONWaitSwitchOffMessage(IN:=FALSE);
	END_IF;

(* Ausgabe ob der Prozesszustand Aktiv ist *)
	T_ExchgParam.T_Visu.xActiveProcessState_St1St2:=	(T_NovRam.T_Parameter.T_PartAnalysis[gciStationSt1].sFileName <> '') OR (T_NovRam.T_Parameter.T_PartAnalysis[gciStationSt1].diActual_NumberHoleToWork <> 0);
	TProcess.T_Ctrle.xActiveProcessState:=T_ExchgParam.T_Visu.xActiveProcessState_St1St2;

(* Ausgabe der abgelaufenen Automat Prozesszeit *)
T_ExchgParam.T_StationCommon.T_Param_Machine.T_ParamAutomat.tAutoProcessTime_St1St2:=
										T_NovRam.T_Parameter.T_Machine.T_ParamAutomat.tAutoProcessTime_St1St2;
T_ExchgParam.T_StationCommon.T_Param_Machine.T_ParamAutomat.iAutoProcessDay_St1St2:=
										T_NovRam.T_Parameter.T_Machine.T_ParamAutomat.iAutoProcessDay_St1St2;

(* Ausgabe der Anzahl bearbeitenden Wstk *)
T_ExchgParam.T_StationCommon.T_Param_Machine.T_ParamAutomat.diNumberPartWorked_St1St2:=
										T_NovRam.T_Parameter.T_Machine.T_ParamAutomat.diNumberPartWorked_St1St2;

(* Eingabe WzWechsel *)
IF (T_ExchgParam.T_SafetyCtrl.bStateMessageRequest <> 0) THEN
	IF T_ExchgParam.T_SafetyCtrl.xSelect_ToolChange_St1 THEN
		T_ExchgParam.T_SafetyCtrl.xSelect_ToolChange_St1:=FALSE;
		IF (T_ExchgParam.T_SafetyCtrl.bState_Select_St1 = 0) THEN
			T_ExchgParam.T_SafetyCtrl.bState_Select_St1:=1;
		ELSIF (T_ExchgParam.T_SafetyCtrl.bState_Select_St1 = 1) THEN
			T_ExchgParam.T_SafetyCtrl.bState_Select_St1:=0;
		END_IF;
	END_IF;
ELSE
	T_ExchgParam.T_SafetyCtrl.bState_Select_St1:=0;
	T_ExchgParam.T_SafetyCtrl.xSelect_ToolChange_St1:=FALSE;
END_IF;

T_ExchgParam.T_StationCommon.T_Param_StationWork.T_TorqueSystem.rActual_Torque:=T_NovRam.T_Parameter.T_StationWork[1].T_TorqueSystem.rActual_Torque;
T_ExchgParam.T_StationCommon.T_Param_StationWork.T_TorqueSystem_L.rActual_Torque:=T_NovRam.T_Parameter.T_StationWork[1].T_TorqueSystem_L.rActual_Torque;
T_ExchgParam.T_StationCommon.T_Param_StationWork.T_TorqueSystem_M.rActual_Torque:=T_NovRam.T_Parameter.T_StationWork[1].T_TorqueSystem_M.rActual_Torque;
END_ACTION
ACTION CtrlSetupKeySwitch:
(* Ctrl SecurityKey-->Switch from NormalOperate to SetupOperate or SetupOperate to NormalOperate *)
	xTmp:=	NOT(xChangePage)
			(*AND T_Visu.T_CtrleAction.xDone*)
			AND NOT(T_Visu.T_CtrleAction.xExecute);
	RisingEdgeSpecialLayer(CLK:=xSecurityKey);
	FallingEdgeSpecialLayer(CLK:=xSecurityKey);
	IF xTmp THEN
		IF RisingEdgeSpecialLayer.Q THEN
			iSaveSetupMode:=iSetupMode;
			T_Visu.T_CtrleAction.iFunction:=2;
			T_Visu.T_CtrleAction.xExecute:=TRUE;
		END_IF;
		IF FallingEdgeSpecialLayer.Q THEN
			T_Visu.T_CtrleAction.iFunction:=1;
			T_Visu.T_CtrleAction.xExecute:=TRUE;
		END_IF;
	END_IF;
(* Check if the State from NormalOperate to SetupOperate or SetupOperate to NormalOperate has changed *)
	IF NOT(xFct_GetNormalOperateActive(dwActualPage:=T_Visu.T_PlcParam.dwActualPage)) AND NOT(xFct_GetSetupOperateActive(dwActualPage:=T_Visu.T_PlcParam.dwActualPage)) THEN
		(* Disable the force of set to a OperateMode *)
		xForceSetupOperate:=FALSE;
		xForceNormalOperate:=FALSE;
	END_IF;
	IF xSecurityKey AND xFct_GetNormalOperateActive(dwActualPage:=T_Visu.T_PlcParam.dwActualPage) THEN
		xForceSetupOperate:=TRUE;
	END_IF;
	IF xSecurityKey AND xFct_GetSetupOperateActive(dwActualPage:=T_Visu.T_PlcParam.dwActualPage) THEN
		xForceSetupOperate:=FALSE;
		xForceNormalOperate:=FALSE;
	END_IF;
	IF NOT(xSecurityKey) AND xFct_GetSetupOperateActive(dwActualPage:=T_Visu.T_PlcParam.dwActualPage) THEN
		xForceNormalOperate:=TRUE;
	END_IF;
	IF NOT(xSecurityKey) AND xFct_GetNormalOperateActive(dwActualPage:=T_Visu.T_PlcParam.dwActualPage) THEN
		xForceSetupOperate:=FALSE;
		xForceNormalOperate:=FALSE;
	END_IF;
	IF xForceNormalOperate OR xForceSetupOperate THEN
		TONWaitForceChangeOperateMode(IN:=TRUE,PT:=T#0.2s);
		IF TONWaitForceChangeOperateMode.Q THEN
				iTestCounter:=iTestCounter+1;
				TONWaitForceChangeOperateMode(IN:=FALSE);
				xTmp:=	NOT(xChangePage)
						AND T_Visu.T_CtrleAction.xDone
						AND NOT(T_Visu.T_CtrleAction.xExecute);
				IF xTmp THEN
					IF xForceNormalOperate THEN
						T_Visu.T_CtrleAction.iFunction:=1;
					END_IF;
					IF xForceSetupOperate THEN
						iSaveSetupMode:=iSetupMode;
						T_Visu.T_CtrleAction.iFunction:=2;
					END_IF;
					T_Visu.T_CtrleAction.xExecute:=TRUE;
				END_IF;
		END_IF;
	ELSE
		TONWaitForceChangeOperateMode(IN:=FALSE);
	END_IF;
END_ACTION
ACTION CtrlSetupOperateModeSwitch:
(* Ctrl SetupOperateModeSwitch --> switch from one SetupOperate Mode to the other *)
	xTmp:=	NOT(xChangePage)
			AND T_Visu.T_CtrleAction.xDone
			AND NOT(T_Visu.T_CtrleAction.xExecute);
	IF xTmp THEN
		RisingEdgeSetupMode(CLK:=(iSaveSetupMode <> iSetupMode));
		IF (T_ExchgParam.T_Visu.bActiveSetupMode <> 0) THEN
			IF RisingEdgeSetupMode.Q THEN
				iSaveSetupMode:=iSetupMode;
				T_Visu.T_CtrleAction.iFunction:=2;
				T_Visu.T_CtrleAction.xExecute:=TRUE;
			END_IF;
		ELSE
			iSaveSetupMode:=iSetupMode;
		END_IF;
	END_IF;
(* Check if the State of the SetupMode has changed *)
	IF xFct_GetSetupOperateActive(dwActualPage:=T_Visu.T_PlcParam.dwActualPage) THEN
		IF (iSetupMode = 1) AND xFct_GetSetupMode(dwActualPage:=T_Visu.T_PlcParam.dwActualPage, iSetupModeRequest:=1) THEN
			(* Disable the force of set to a SetupMode *)
			xForceSetupMode:=FALSE;
		END_IF;
		IF (iSetupMode = 2) AND xFct_GetSetupMode(dwActualPage:=T_Visu.T_PlcParam.dwActualPage, iSetupModeRequest:=2) THEN
			(* Disable the force of set to a SetupMode *)
			xForceSetupMode:=FALSE;
		END_IF;
		IF (iSetupMode = 1) AND NOT(xFct_GetSetupMode(dwActualPage:=T_Visu.T_PlcParam.dwActualPage, iSetupModeRequest:=1)) THEN
			xForceSetupMode:=TRUE;
		END_IF;
		IF (iSetupMode = 2) AND NOT(xFct_GetSetupMode(dwActualPage:=T_Visu.T_PlcParam.dwActualPage, iSetupModeRequest:=2)) THEN
			xForceSetupMode:=TRUE;
		END_IF;

		IF xForceSetupMode THEN
			TONWaitForceChangeSetupMode(IN:=TRUE,PT:=T#0.2s);
			IF TONWaitForceChangeSetupMode.Q THEN
					iTestCounter1:=iTestCounter1+1;
					TONWaitForceChangeSetupMode(IN:=FALSE);
					xTmp:=	NOT(xChangePage)
							AND T_Visu.T_CtrleAction.xDone
							AND NOT(T_Visu.T_CtrleAction.xExecute);
					IF xTmp THEN
						IF xForceSetupMode THEN
							iSaveSetupMode:=iSetupMode;
							T_Visu.T_CtrleAction.iFunction:=2;
						END_IF;
						T_Visu.T_CtrleAction.xExecute:=TRUE;
					END_IF;
			END_IF;
		ELSE
			TONWaitForceChangeSetupMode(IN:=FALSE);
		END_IF;
	ELSE
		TONWaitForceChangeSetupMode(IN:=FALSE);
	END_IF;
END_ACTION
ACTION CtrlSpindleTime:
(* Gilt für die Aufzeichnung der Dauer der Spindelrotation *)
CASE T_ExchgParam.bToolSpindleActive OF
1:	(* Maxon Spindel *)
	T_ExchgParam.T_StationCommon.iSpindelActiveRotationDay:=TStation_Work_St1.THWWorkStation.TCtrlWork.iSpindelActiveRotationDay;
	T_ExchgParam.T_StationCommon.tSpindelActiveRotationTime:=TStation_Work_St1.THWWorkStation.TCtrlWork.tSpindelActiveRotationTime;
2:	(* Beckhoff Spindel L *)
	T_ExchgParam.T_StationCommon.iSpindelActiveRotationDay:=TStation_Work_St1.THWWorkStation.TCtrlWork.iSpindel2ActiveRotationDay;
	T_ExchgParam.T_StationCommon.tSpindelActiveRotationTime:=TStation_Work_St1.THWWorkStation.TCtrlWork.tSpindel2ActiveRotationTime;
3:	(* Beckhoff Spindel M *)
	T_ExchgParam.T_StationCommon.iSpindelActiveRotationDay:=TStation_Work_St1.THWWorkStation.TCtrlWork.iSpindel3ActiveRotationDay;
	T_ExchgParam.T_StationCommon.tSpindelActiveRotationTime:=TStation_Work_St1.THWWorkStation.TCtrlWork.tSpindel3ActiveRotationTime;
END_CASE;
IF T_StartUp.T_State.xCompleted THEN
	T_NovRAM.T_Parameter.T_StationWork[1].iSpindelActiveRotationDay:=TStation_Work_St1.THWWorkStation.TCtrlWork.iSpindelActiveRotationDay;
	T_NovRAM.T_Parameter.T_StationWork[1].tSpindelActiveRotationTime:=TStation_Work_St1.THWWorkStation.TCtrlWork.tSpindelActiveRotationTime;
	T_NovRAM.T_Parameter.T_StationWork[1].iSpindel2ActiveRotationDay:=TStation_Work_St1.THWWorkStation.TCtrlWork.iSpindel2ActiveRotationDay;
	T_NovRAM.T_Parameter.T_StationWork[1].tSpindel2ActiveRotationTime:=TStation_Work_St1.THWWorkStation.TCtrlWork.tSpindel2ActiveRotationTime;
	T_NovRAM.T_Parameter.T_StationWork[1].iSpindel3ActiveRotationDay:=TStation_Work_St1.THWWorkStation.TCtrlWork.iSpindel3ActiveRotationDay;
	T_NovRAM.T_Parameter.T_StationWork[1].tSpindel3ActiveRotationTime:=TStation_Work_St1.THWWorkStation.TCtrlWork.tSpindel3ActiveRotationTime;
END_IF;
END_ACTION
ACTION CtrlStartStopButton:
(* Externe StartTaste *)
	xTmp:=	NOT(xChangePage)
			AND T_Visu.T_CtrleAction.xDone
			AND NOT(T_Visu.T_CtrleAction.xExecute)
			AND NOT(T_StartUp.T_State.xBlockChangeMovementVisu)
			AND TProcess.T_Ctrle.xDone;
	IF xTmp THEN
		(* manage rising edge start button *)
		IF xStartButton THEN
			dwSaveVisuPage:=T_Visu.T_PlcParam.dwActualPage;
			CASE T_Visu.T_PlcParam.dwActualPage OF
			gT_PageNumber.iAutoMode_Process, gT_PageNumber.iAutoMode_ProcessValue1, gT_PageNumber.iAutoMode_ProcessValue2, gT_PageNumber.iAutoMode_PartQuality:
					T_Visu.T_CtrleAction.iFunction:=700 + 2;		(* Automat Prozess-->Wstk bearbeiten *)

			gT_PageNumber.iAutoMode_Referencing:			(* Maschinenreferenzierung Prozess *)
					T_Visu.T_CtrleAction.iFunction:=700 + 1;

			gT_PageNumber.iHandMode_Process, gT_PageNumber.iHandMode_WorkParameter, gT_PageNumber.iHandMode_RegulatorPara,
			gT_PageNumber.iHandMode_OnlineChange, gT_PageNumber.iHandMode_ConfigPosition:				(* HandBetrieb Prozess *)
					T_Visu.T_CtrleAction.iFunction:=600 + 3;

			gT_PageNumber.iWorkStation_Axis1:
				(* Abfragen ob die Achse eine Absolute Position oder Geschwindigkeitsbewegung ausführen kann *)
				CASE T_ExchgParam.T_TeachIn.iSetup_AxisSel OF
				gciAxisZ_St1:		T_Visu.T_CtrleAction.iFunction:=210;			(* Absolute Bewegung einer ausgewählten Achse auf ausgewählte Position *)
				gciAxisS_St1,3:	T_Visu.T_CtrleAction.iFunction:=207;			(* Achse Geschwindigkeitsmodus für Spindel *)
				END_CASE;

			gT_PageNumber.iWorkStation_Function1:
					T_Visu.T_CtrleAction.iFunction:=401;			(* Ausführen von Stationsfunktionen der Bearbeitungsstation *)

			gT_PageNumber.iWorkStation_Setup3:
				IF (T_ExchgParam.T_StationCommon.bSelectZAxisProcedure <= 1) THEN
					T_Visu.T_CtrleAction.iFunction:=405;			(* Ausführen von Stationsfunktionen der Bearbeitungsstation für die Einrichtung der Z Achse und des oberen Führungsrohr *)
				ELSE
					T_Visu.T_CtrleAction.iFunction:=402;			(* Ausführen von Stationsfunktionen der Bearbeitungsstation für Ersteinrichtung der Z Achse *)
				END_IF;

			gT_PageNumber.iWorkStation_Setup1:
					T_Visu.T_CtrleAction.iFunction:=403;			(* Ausführen der Stationsfunktion für das Kalibrieren des ToolDefelction und ToolTorque *)

			gT_PageNumber.iWorkStation_Setup2:
					T_Visu.T_CtrleAction.iFunction:=404;			(* Ausführen der Stationsfunktion für den BurnIn der Spindeln über ausgewählte Stationen *)

			END_CASE;
			T_Visu.T_CtrleAction.xExecute:=TRUE;
			iSaveStartedVisuFunction_St1St2:=T_Visu.T_CtrleAction.iFunction;
		END_IF;
	END_IF;

	xTmp:=	NOT(T_Visu.T_CtrleAction.xExecute) AND T_Visu.T_CtrleAction.xDone AND
			NOT(T_Visu.T_CtrleProcess.xExecute) AND T_Visu.T_CtrleProcess.xDone AND
			NOT(xTmpStationSetupAxisZFunction) AND NOT(xTmpStationSetupAxisZFunctionToolGuide) AND
			TProcess.T_Ctrle.xDone;
	IF xTmp THEN
		iSaveStartedVisuFunction_St1St2:=0;
	END_IF;
(* Externe StoppTaste *)
	xTmp:=	NOT(T_Visu.T_CtrleAction.xExecute);
	IF xStopButton AND xTmp THEN
		T_Visu.T_CtrleAction.iFunction:=0;
		IF (NOT(TProcess.T_Ctrle.xDone) AND NOT(TProcess.T_Ctrle.xError)) THEN
			(* Prozess ist aktiv *)
			IF (iSaveStartedVisuFunction_St1St2 >= 600) AND (iSaveStartedVisuFunction_St1St2 <= 698) THEN
				(* Prozess welches im HandBetrieb aktiviert wurde, ist aktiv *)
				T_Visu.T_CtrleAction.iFunction:=699;
			END_IF;
			IF (iSaveStartedVisuFunction_St1St2 >= 700) AND (iSaveStartedVisuFunction_St1St2 <= 796) THEN
				IF (T_ExchgParam.T_Visu.T_Message.iState <> 110) THEN	(* Aufforderung: Leerfahren aktivieren <StartTaste>, abbr. <StopTaste> ? *)
					(* Prozess welches im Automat aktiviert wurde, ist aktiv *)
					T_Visu.T_CtrleAction.iFunction:=799;
				END_IF;
			END_IF;
		ELSE
			(* Prozess ist nicht Aktiv *)
			IF ((iSaveStartedVisuFunction_St1St2 >= 400) AND (iSaveStartedVisuFunction_St1St2 <= 496)) OR
			    (T_Visu.T_CtrleAction.xFunctionActive AND (T_Visu.T_PlcParam.dwActualPage <> gT_PageNumber.iWorkStation_Axis1)) THEN
				(* Stationsfunktion muss gestoppt werden *)
				T_Visu.T_CtrleAction.iFunction:=499;
			ELSE
				(* Prozess und Stationsfunktionen sind nicht Aktiv-->Achsen stoppen *)
				CASE T_Visu.T_PlcParam.dwActualPage OF
				gT_PageNumber.iWorkStation_Axis1:
					T_Visu.T_CtrleAction.iFunction:=202;
				gT_PageNumber.iAutoMode_ToolChange:
					T_Visu.T_CtrleAction.iFunction:=201;
				END_CASE;
			END_IF;
		END_IF;
		IF (T_Visu.T_CtrleAction.iFunction <> 0) THEN
			T_Visu.T_CtrleAction.xExecute:=TRUE;
		END_IF;
	END_IF;
END_ACTION
ACTION CtrlTaskBar:
(* Bt navigation panel *)
	xTmp:=	NOT(xChangePage)
			AND T_Visu.T_CtrleAction.xDone
			AND NOT(T_Visu.T_CtrleAction.xExecute)
			AND NOT(T_StartUp.T_State.xBlockChangeMovementVisu);
	IF xTmp THEN
		RisingEdgeTouchScreenNavPanel(CLK:=		(T_ExchgParam.T_TouchScreenNavPanel.wActivBt
												AND T_ConfigPage.wMaskTouchScreenNavPanel) <> 16#0);
		(* check if more than one button is pressed-->if only one Button than start the procedure *)
		IF xFct_CheckSingleButtonActivation(wInputButton:=T_ExchgParam.T_TouchScreenNavPanel.wActivBt) THEN
		(* activ action of rising edge *)
			IF RisingEdgeTouchScreenNavPanel.Q THEN
				IF xFct_GetParameterPageActive(dwActualPage:=T_Visu.T_PlcParam.dwActualPage) THEN
					(* Do not change the page, if the Parameter page is active-->change only the Task *)
					awSaveStateTaskBar[T_ExchgParam.T_Visu.bActiveSetupMode]:=T_ExchgParam.T_TouchScreenNavPanel.wActivBt;
					ii:=iFct_GetBitNumber(wInputButton:=T_ExchgParam.T_TouchScreenNavPanel.wActivBt);
					(* Da diese Software keine Parameterlisten bezogen auf Task hat, sind alle gleichgestellt und muss beim Taskwechsel nicht mehr ein Update Parameter durchgeführt werden *)
					(*
					xUpdateStationParameter:=TRUE;
					*)
				ELSE
					ii:=iFct_GetBitNumber(wInputButton:=T_ExchgParam.T_TouchScreenNavPanel.wActivBt);
					IF (T_ConfigPage.aiRTrigActionTouchScreenNavPanel[ii,1] <> 0) THEN
						T_Visu.T_CtrleAction.iFunction:=10000 + DWORD_TO_INT(dwSaveActualPageTask[T_ExchgParam.T_Visu.bActiveSetupMode,ii]);
						T_Visu.T_CtrleAction.xExecute:=TRUE;
					END_IF;
					awSaveStateTaskBar[T_ExchgParam.T_Visu.bActiveSetupMode]:=T_ExchgParam.T_TouchScreenNavPanel.wActivBt;
				END_IF;
			END_IF;
		END_IF;
		T_ExchgParam.T_TouchScreenNavPanel.wActivBt:=0;
	ELSE
		T_ExchgParam.T_TouchScreenNavPanel.wActivBt:=0;
		(* Init. rising and falling edge *)
		RisingEdgeTouchScreenNavPanel(CLK:=FALSE);
	END_IF
END_ACTION
ACTION CtrlVisuFunction:
(* waiting for executing action *)
	(* ...monitor Key panel "Enter" *)
	RisingEdgeKeyPanel_Enter(CLK:=T_ExchgParam.T_Visu.xKey_Enter);
	(* ...monitor Key panel "Esc" *)
	RisingEdgeKeyPanel_Esc(CLK:=T_ExchgParam.T_Visu.xKey_Escape);
	(*... not ready *)
	TimerNotReady(IN:=FALSE, PT:=T#2s);
	T_Visu.T_CtrleAction.xNotReady:=TimerNotReady.Q;
	(* ...message *)
	RisingEdgeActionNotReady(CLK:=T_Visu.T_CtrleAction.xNotReady);
	IF RisingEdgeActionNotReady.Q AND T_ExchgParam.T_Visu.T_Message.iState < 350 THEN
		T_ExchgParam.T_Visu.T_Message.iState:=201;	(* Warnung: Nicht bereit auszuführen ! *)
	END_IF
	(* Release 'Not ready' action control structure *)
	FallingEdgeActionNotReady(CLK:=T_Visu.T_CtrleAction.xNotReady);
	IF FallingEdgeActionNotReady.Q THEN
		T_Visu.T_CtrleAction.xExecute:=FALSE;
		T_Visu.T_CtrleAction.xDone:=TRUE;
		T_Visu.T_CtrleAction.xErr:=FALSE;
		T_Visu.T_CtrleAction.udiErrorID:=0;
		iStepAction:=1;
		iStepActionRef:=1;
		iStepActionNovRam:=1;
		xStepActionDone:=FALSE;
		TimerAction(IN:=FALSE);
	END_IF
	(* ...done *)
	RisingEdgeActionDone(CLK:=T_Visu.T_CtrleAction.xDone);
	IF RisingEdgeActionDone.Q THEN
		IF (T_ExchgParam.T_Visu.T_Message.iState = 0) AND NOT(xBlockConfirmMessage) THEN
			T_ExchgParam.T_Visu.T_Message.iState:=32;	(* Info: Aktion beendet ! *)
		END_IF
		xBlockConfirmMessage:=FALSE;
	END_IF
	(* ...error *)
	RisingEdgeActionError(CLK:=T_Visu.T_CtrleAction.xErr);
	IF RisingEdgeActionError.Q THEN
	(* call function bloc action error *)
		(* Init. variable *)
		T_Visu.T_CtrleAction.xExecute:=FALSE;
		T_Visu.T_CtrleAction.xDone:=TRUE;
		T_Visu.T_CtrleAction.xErr:=FALSE;
		T_Visu.T_CtrleAction.xNotReady:=FALSE;
		T_Visu.T_CtrleAction.udiErrorID:=0;
		iStepAction:=1;
		iStepActionNovRam:=1;
		iStepActionRef:=1;
		xStepActionDone:=FALSE;
	END_IF
	(* ...reset *)
	RisingEdgeResetAction(CLK:=T_Visu.T_CtrleAction.xReset);
	IF RisingEdgeResetAction.Q THEN
		(* Init. variable *)
		T_Visu.T_CtrleAction.xExecute:=FALSE;
		T_Visu.T_CtrleAction.xDone:=TRUE;
		T_Visu.T_CtrleAction.xErr:=FALSE;
		T_Visu.T_CtrleAction.xNotReady:=FALSE;
		T_Visu.T_CtrleAction.udiErrorID:=0;
		iStepAction:=1;
		iStepActionNovRam:=1;
		iStepActionRef:=1;
		xStepActionDone:=FALSE;
		TimerAction(IN:=FALSE);
		(* Release reset *)
		T_Visu.T_CtrleAction.xReset:=FALSE;
	END_IF
	(* Ausgabe der Zeilen Meldungen *)
	IF (T_ExchgParam.T_Visu.T_Message.iState >= 1) AND (T_ExchgParam.T_Visu.T_Message.iState <= 100) THEN
		T_ExchgParam.T_Visu.T_Message.xShowMessageInfo:=TRUE;
		T_ExchgParam.T_SafetyCtrl.xHideSafetyCtrlMessage:=TRUE;
	ELSE T_ExchgParam.T_Visu.T_Message.xShowMessageInfo:=FALSE; END_IF;
	IF (T_ExchgParam.T_Visu.T_Message.iState >= 101) AND (T_ExchgParam.T_Visu.T_Message.iState <= 200) THEN
		T_ExchgParam.T_Visu.T_Message.xShowMessageInput:=TRUE;
		T_ExchgParam.T_SafetyCtrl.xHideSafetyCtrlMessage:=TRUE;
	ELSE T_ExchgParam.T_Visu.T_Message.xShowMessageInput:=FALSE; END_IF;
	IF (T_ExchgParam.T_Visu.T_Message.iState >= 201) AND (T_ExchgParam.T_Visu.T_Message.iState <= 350) THEN
		T_ExchgParam.T_Visu.T_Message.xShowMessageWarning:=TRUE;
		T_ExchgParam.T_SafetyCtrl.xHideSafetyCtrlMessage:=TRUE;
	ELSE T_ExchgParam.T_Visu.T_Message.xShowMessageWarning:=FALSE; END_IF;
	(* Ausblenden der Zeilen Meldungen *)
	CASE iStepShowMessage OF
	1:	IF ((T_ExchgParam.T_Visu.T_Message.iState >= 1) AND (T_ExchgParam.T_Visu.T_Message.iState <= 100)) OR
		     ((T_ExchgParam.T_Visu.T_Message.iState >= 201) AND (T_ExchgParam.T_Visu.T_Message.iState <= 350)) THEN
			(* Dies gilt für Info und Warnungsmeldung *)
			iSaveMessage:=T_ExchgParam.T_Visu.T_Message.iState;
			iStepShowMessage:=iStepShowMessage + 1;
			TONWaitShowMessage(IN:=FALSE);
		END_IF;
	2:	IF T_StartUp.T_State.xCompleted OR (T_ExchgParam.T_Visu.T_Message.iState =225) OR (T_ExchgParam.T_Visu.T_Message.iState = 226) THEN
			TONWaitShowMessage(IN:=TRUE,PT:=T#3s);
		ELSE
			TONWaitShowMessage(IN:=TRUE,PT:=T#0.5s);
		END_IF;
		IF TONWaitShowMessage.Q THEN
			T_ExchgParam.T_Visu.T_Message.iState:=0;	(* Meldung löschen *)
			iStepShowMessage:=1;
		END_IF;
		(* Überprüfe ob nicht die Aktuelle Meldung überschrieben wurde *)
		IF (iSaveMessage <> T_ExchgParam.T_Visu.T_Message.iState) THEN
			iSaveMessage:=T_ExchgParam.T_Visu.T_Message.iState;
			iStepShowMessage:=1;	(* Erneute Ausgabe für neue Meldung mit der gleichen Anzeige Zeit *)
		END_IF;
	ELSE
		iStepShowMessage:=1;
	END_CASE;

	RisingEdgeExecuteAction(CLK:=T_Visu.T_CtrleAction.xExecute);
	IF RisingEdgeExecuteAction.Q THEN
		(* confirm action execution *)
		IF (NOT(T_StartUp.T_State.xBlockChangeMovementVisu) OR (T_Visu.T_CtrleAction.iFunction = 499)) AND
		     NOT(xTmpProcMachineStop)  THEN
			T_Visu.T_CtrleAction.xDeleteVisuFunction:=TRUE;
			CtrlVisuFunctionDelete;
		END_IF;
		T_Visu.T_CtrleAction.xExecute:=FALSE;
		CASE T_Visu.T_CtrleAction.iFunction OF
		(* Set NormalOperate *)
		1:	xSetNewPage:=TRUE;
			T_Visu.T_PlcParam.dwSetNewPage:=dwSaveActualPageTask[0,iFct_GetBitNumber(wInputButton:=awSaveStateTaskBar[0])];
			tTimeOutAction:=T#3s;
		(* Set SetupOperate *)
		2:	xSetNewPage:=TRUE;
			iTmpSetupMode:=iSetupMode;
			IF (iTmpSetupMode<1) OR (iTmpSetupMode>3) THEN iTmpSetupMode:=1; END_IF;
			T_Visu.T_PlcParam.dwSetNewPage:=dwSaveActualPageTask[iTmpSetupMode,iFct_GetBitNumber(wInputButton:=awSaveStateTaskBar[iTmpSetupMode])];
			tTimeOutAction:=T#3s;
		(* Set parameter page *)
		3:	xSetParameterPage:=TRUE;
			tTimeOutAction:=T#2s;
		(* Set previous page *)
		5:	xSetPreviousPage:=TRUE;
			tTimeOutAction:=T#3s;
		(* previous  page vertical *)
		11:	xPreviousPageVertical:=TRUE;
			tTimeOutAction:=T#3s;
		(* next page vertical *)
		12:	xNextPageVertical:=TRUE;
			tTimeOutAction:=T#3s;
		(* Löschen der Fehlerliste *)
		97:	xDeleteErrorList:=TRUE;
			tTimeOutAction:=T#5s;

		(* Quittieren des Fehler/Warnung *)
		99:	xResetErrorWarning:=TRUE;
			tTimeOutAction:=T#5s;
		(* LampTest-->Lamp ON/OFF *)
		100:	xLampTestOnOff:=TRUE;
			tTimeOutAction:=T#999999s;
		(* LampTest-->Lamp Blink ON/OFF *)
		101:	xLampTestBlinkOnOff:=TRUE;
			tTimeOutAction:=T#999999s;
		(* LampTest-->LampTest ON *)
		102:	xLampTestActive:=TRUE;
			tTimeOutAction:=T#999999s;

		(* Meldungsfenster Öffnen *)
		104:	xOpenMessageWindow:=TRUE;
			tTimeOutAction:=T#3s;
		(* Maschinen Tür Zuhaltun EIN/AUS *)
		105:	xMachineDoorUpGuardControlTogOnOff:=TRUE;
			tTimeOutAction:=T#5s;

		(* Ändern des Operator Passwortes *)
		110:	xChangeOperatorPassword:=TRUE;
			tTimeOutAction:=T#20s;

		(* Umschalten Z Ink Wert für Bearbeitung *)
		113:xSelectZInkWorkInfo:=TRUE;
			tTimeOutAction:=T#5s;
		(* Umschalten Z Ink Wert für Zentrierung *)
		114:xSelectZInkCentringInfo:=TRUE;
			tTimeOutAction:=T#5s;

		(* Resetten des Werkzeugwechsel für den Automatik für Station 1-->braucht mindestens den OperatorLevel *)
		115:	xProcessStation1ResetToolChange:=TRUE;
			tTimeOutAction:=T#5s;
		(* Z Achse auf WzWechsel Pos setzen *)
		116:	xZAxisMoveToToolChangePos:=TRUE;
			tTimeOutAction:=T#5s;
			ptrTCommonAxisActive:=ptrTAxisZ_St1;
			rZAxisSelectPosition:=T_NovRAM.T_Parameter.T_StationWork[1].T_StProcess.rPositionToolChange;
			ptrTCommonAxisActive^.T_CtrleSingle.lrVelocity:=gcarAxisConfig[1].rPositionSpeed;
		(* Z Achse auf LadePos setzen *)
		117: xZAxisMoveToLoadPos:=TRUE;
			tTimeOutAction:=T#5s;
			ptrTCommonAxisActive:=ptrTAxisZ_St1;
			rZAxisSelectPosition:=grZ_LoadPos;
			ptrTCommonAxisActive^.T_CtrleSingle.lrVelocity:=gcarAxisConfig[1].rPositionSpeed;
		(* Speichern Z EndPos Berechnet *)
		118:	xZSaveEndPosCalc:=TRUE;
			tTimeOutAction:=T#5s;

		(* OnlineChange Parameter ToolTorque Drehmoment Schwellwert HC + *)
		120:	xOnlineChange_TorqueLevelHCMore:=TRUE;
			tTimeOutAction:=T#3s;
		(* OnlineChange Parameter ToolTorque Drehmoment Schwellwert HC - *)
		121:	xOnlineChange_TorqueLevelHCLess:=TRUE;
			tTimeOutAction:=T#3s;

		(* OnlineChange Parameter Zylinder ToolDeflection Auslenkkraft + *)
		126:	xOnlineChange_DeflectionForceMore:=TRUE;
			tTimeOutAction:=T#3s;
		(* OnlineChange Parameter Zylinder ToolDeflection Auslenkkraft - *)
		127:	xOnlineChange_DeflectionForceLess:=TRUE;
			tTimeOutAction:=T#3s;
		(* OnlineChange Parameter Z Achse Bearbeitungsgeschwindigkeit vorwärts + *)
		128:	xOnlineChange_Z_ForwardSpeedMore:=TRUE;
			tTimeOutAction:=T#3s;
		(* OnlineChange Parameter Z Achse Bearbeitungsgeschwindigkeit vorwärts - *)
		129:	xOnlineChange_Z_ForwardSpeedLess:=TRUE;
			tTimeOutAction:=T#3s;
		(* OnlineChange Parameter Z Achse Bearbeitungsgeschwindigkeit rückwärts + *)
		130:	xOnlineChange_Z_BackwardSpeedMore:=TRUE;
			tTimeOutAction:=T#3s;
		(* OnlineChange Parameter Z Achse Bearbeitungsgeschwindigkeit rückwärts - *)
		131:	xOnlineChange_Z_BackwardSpeedLess:=TRUE;
			tTimeOutAction:=T#3s;
		(* OnlineChange Parameter Z Achse rückwärts Offset + *)
		132:	xOnlineChange_Z_BackwardOffsetMore:=TRUE;
			tTimeOutAction:=T#3s;
		(* OnlineChange Parameter Z Achse rückwärts Offset - *)
		133:	xOnlineChange_Z_BackwardOffsetLess:=TRUE;
			tTimeOutAction:=T#3s;
		(* OnlineChange Parameter S Achse Bearbeitungsgeschwindigkeit + *)
		134:	xOnlineChange_S_WorkSpeedMore:=TRUE;
			tTimeOutAction:=T#3s;
		(* OnlineChange Parameter S Achse Bearbeitungsgeschwindigkeit - *)
		135:	xOnlineChange_S_WorkSpeedLess:=TRUE;
			tTimeOutAction:=T#3s;

		(* Löschen des Prozesszustandspeicher *)
		150:	xDeleteProcessState:=TRUE;
			tTimeOutAction:=T#5s;
		(* Endlos Prozess EIN/AUS *)
		151:	xEndlessProcessOnOff:=TRUE;
			tTimeOutAction:=T#5s;
		(* Zentrieren EIN/AUS *)
		152:	xCentringONOFF:=TRUE;
			tTimeOutAction:=T#5s;
		(* NurZentrieren EIN/AUS *)
		153:	xOnlyCentringONOFF:=TRUE;
			tTimeOutAction:=T#5s;
		(* Suspension EIN/AUS *)
		154:	xSuspensionONOFF:=TRUE;
			tTimeOutAction:=T#5s;
		(* ZylWPUnfix EIN/AUS *)
		155:	xCylWPUnfixONOFF:=TRUE;
			tTimeOutAction:=T#5s;

		(* Setup Potentiometer *)
		170:	xSetupPotentiometer:=TRUE;
			tTimeOutAction:=T#0s;
		(* Torque Offset - *)
		171:	xTorqueOffsetMinus:=TRUE;
			tTimeOutAction:=T#0s;
		(* Torque Offset + *)
		172:	xTorqueOffsetPlus:=TRUE;
			tTimeOutAction:=T#0s;
		(* Save Torque Scale *)
		173:	xSaveTorqueScale:=TRUE;
			tTimeOutAction:=T#5s;
		(* Save Torque Position *)
		174:	xSaveTorquePosition:=TRUE;
			tTimeOutAction:=T#5s;

		(* Auswahl Position Führungsrohr *)
		181:	xSelectConfigPosition_1:=TRUE;
			tTimeOutAction:=T#3s;
		(* Auswahl Abstand Führungsrohr *)
		182:	xSelectConfigPosition_2:=TRUE;
			tTimeOutAction:=T#3s;
		(* Auswahl Werkzeug *)
		183:	xSelectConfigPosition_3:=TRUE;
			tTimeOutAction:=T#3s;
		(* Auswahl Führungsrohreinsatz *)
		184:	xSelectConfigPosition_4:=TRUE;
			tTimeOutAction:=T#3s;
		(* KonfigPos EIN/AUS *)
		185:	xConfigPosOnOff:=TRUE;
			tTimeOutAction:=T#5s;
		(* Speichern der Positionskonfiguration *)
		186:	xSaveConfigPosition:=TRUE;
			tTimeOutAction:=T#5s;

		(* Konventioneller Regler *)
		190:	xRegulatorType1:=TRUE;
			tTimeOutAction:=T#5s;
		(* Adaptive Voschub Regler *)
		191:	xRegulatorType2:=TRUE;
			tTimeOutAction:=T#5s;
		(* Konventioneller PD Regler *)
		192:	xRegulatorType3:=TRUE;
			tTimeOutAction:=T#5s;
		(* Regler Parameter speichern *)
		195:	xRegulatorOverlaySave:=TRUE;
			tTimeOutAction:=T#5s;

		(* Spindelkalibrierung EIN/AUS *)
		198:	xSpindelCalibrationONOFF:=TRUE;
			tTimeOutAction:=T#5s;

		200..299:
			CASE T_Visu.T_CtrleAction.iFunction OF
				(* Bewegung einer Achse stoppen *)
				201:	xAxisStop:=TRUE;
					tTimeOutAction:=T#3s;
				(* Bewegung aller Achse stoppen *)
				202:	xAxisStopAll:=TRUE;
					tTimeOutAction:=T#3s;
				(* Achsen Drehmoment Ein/Aus Toggeln *)
				203:	xAxisTogglePower:=TRUE;
					tTimeOutAction:=T#3s;
				(* Achse Resetten *)
				204:	xAxisReset:=TRUE;
					tTimeOutAction:=T#3s;
				(* Achse Geschwindigkeitsmodus *)
				207:	xAxisMoveContinous:=TRUE;
					tTimeOutAction:=T#5s;
					CASE T_ExchgParam.T_TeachIn.iSetup_AxisSel OF
					2,3:	ptrTCommonAxisActive:=ptrTAxisS_St1;
					END_CASE;
					ptrTCommonAxisActive^.T_CtrleSingle.lrVelocity:=TCommonTeachParameter.rPositionSpeed;
				(* Achse Absolute Positionsbewegung *)
				210:	xAxisMoveAbsolut:=TRUE;
					tTimeOutAction:=T#999s;
				(* Achse Teach Position *)
				214:	xAxisTeachPosition:=TRUE;
					tTimeOutAction:=T#5s;
				(* Achse Jog/Ink Bewegung +/++ mit Joystick *)
				216:	tTimeOutAction:=T#999s;
					IF xActive_Joystick THEN
						ptrTCommonAxisActive:=ptrTAxisZ_St1;
						ptrTCommonAxisActive^.T_CtrleSingle.lrVelocity:=T_ExchgParam.T_TeachIn.arTeachSelVel[gciAxisZ_St1];
						ptrTCommonAxisActive^.T_CtrleSingle.lrDistance:=T_ExchgParam.T_TeachIn.arTeachSelStep[gciAxisZ_St1];
					ELSE
						ptrTCommonAxisActive:=ptrTCommonAxis;
						ptrTCommonAxisActive^.T_CtrleSingle.lrVelocity:=TCommonTeachParameter.rVelFast;
						ptrTCommonAxisActive^.T_CtrleSingle.lrDistance:=TCommonTeachParameter.rIncFast;
					END_IF;
					IF T_ExchgParam.T_TeachIn.xJogInc_Common_Setup_Axis THEN
						(* Jog Mode *)
						xAxisMoveContinous:=TRUE;
					ELSE
						(* Ink Mode *)
						xAxisMoveRelative:=TRUE;
					END_IF;
				(* Achse Jog/Ink Bewegung -/- - mit Joystick *)
				217:	tTimeOutAction:=T#999s;
					IF xActive_Joystick THEN
						ptrTCommonAxisActive:=ptrTAxisZ_St1;
						IF T_ExchgParam.T_TeachIn.xJogInc_Common_Setup_Axis THEN
							ptrTCommonAxisActive^.T_CtrleSingle.lrVelocity:=T_ExchgParam.T_TeachIn.arTeachSelVel[gciAxisZ_St1] * -1.0;
						ELSE
							ptrTCommonAxisActive^.T_CtrleSingle.lrVelocity:=T_ExchgParam.T_TeachIn.arTeachSelVel[gciAxisZ_St1];
							ptrTCommonAxisActive^.T_CtrleSingle.lrDistance:=T_ExchgParam.T_TeachIn.arTeachSelStep[gciAxisZ_St1] * -1.0;
						END_IF;
					ELSE
						ptrTCommonAxisActive:=ptrTCommonAxis;
						IF T_ExchgParam.T_TeachIn.xJogInc_Common_Setup_Axis THEN
							ptrTCommonAxisActive^.T_CtrleSingle.lrVelocity:=TCommonTeachParameter.rVelFast * -1.0;
						ELSE
							ptrTCommonAxisActive^.T_CtrleSingle.lrVelocity:=TCommonTeachParameter.rVelFast;
							ptrTCommonAxisActive^.T_CtrleSingle.lrDistance:=TCommonTeachParameter.rIncFast * -1.0;
						END_IF;
					END_IF;
					IF T_ExchgParam.T_TeachIn.xJogInc_Common_Setup_Axis THEN
						(* Jog Mode *)
						xAxisMoveContinous:=TRUE;
					ELSE
						(* Ink Mode *)
						xAxisMoveRelative:=TRUE;
					END_IF;
				(* Löschen der berechnete Wert für Wippe des Drehmoment Detection *)
				230:	xResetRockerValue:=TRUE;
					tTimeOutAction:=T#2s;
			END_CASE;
		(* Analogen Wert für Servoventil setzen *)
		300:	xCylSetServoAnalogValue:=TRUE;
			tTimeOutAction:=T#3s;
		(* Zylinder/Ventile Ein/Aus Toggeln *)
		301:	xCylValveToggleOnOff:=TRUE;
			tTimeOutAction:=T#3s;
		(* Zylinder Drucklos schalten *)
		302:	xCylPressurelessON:=TRUE;
			tTimeOutAction:=T#3s;
		(* Zyl WzDrehmoment EIN/AUS *)
		303:	xCylTorqueOnOff:=TRUE;
			tTimeOutAction:=T#3s;
		(* Zyl WzDrehmomentÜberlast EIN/AUS *)
		304:	xCylTorqueOverloadOnOff:=TRUE;
			tTimeOutAction:=T#3s;
		(* Ausführen von Stationsfunktionen der Bearbeitungsstation *)
		401:		xStationWorkFunction:=TRUE;
				tTimeOutAction:=T#0s;
		(* Ausführen von Stationsfunktionen der Bearbeitungsstation für Ersteinrichtung der Z Achse *)
		402:		xStationSetupAxisZFunction:=TRUE;
				tTimeOutAction:=T#0s;
		(* Ausführen der Stationsfunktion für das Kalibrieren des ToolDefelction und ToolTorque *)
		403:		xStationToolCalibrateFunction:=TRUE;
				tTimeOutAction:=T#0s;
		(* Ausführen der Stationsfunktion für den BurnIn der Spindeln über ausgewählte Stationen *)
		404:		xStationSpindleBurnInFunction:=TRUE;
				tTimeOutAction:=T#0s;
		(* Ausführen von Stationsfunktionen der Bearbeitungsstation für Einrichtung der Z Achse und oberes Führungsrohr *)
		405:		xStationSetupAxisZFunctionToolGuide:=TRUE;
				tTimeOutAction:=T#0s;
		(* Stoppen von Stationsfunktionen der rechten Arbeitsstation *)
		497:		xStationStopWorkRight:=TRUE;
				tTimeOutAction:=T#0s;
		(* Stoppen von Stationsfunktionen *)
		499:		xStationStop:=TRUE;
				xStationWorkFunction:=xStationToolCalibrateFunction:=xStationSpindleBurnInFunction:=FALSE;
				xTmpStationSetupAxisZFunction:=xTmpStationSetupAxisZFunctionToolGuide:=FALSE;
				tTimeOutAction:=T#0s;
		(* Prozesse die aus der Stationsebene ausgelöst werden *)
		600..698:	TProcess.T_Ctrle.iFunctNr:=T_Visu.T_CtrleAction.iFunction - 600;
				xActionProcStation:=TRUE;
				tTimeOutAction:=T#1s;
		(* Stoppen vom Prozess welches über den HandBetrieb ausgelöst wurde *)
		699:		xProcStationStop:=TRUE;
				tTimeOutAction:=T#0s;
		(* Prozesse die aus der Maschinenebene ausgelöst werden *)
		701..796:	TProcess.T_Ctrle.iFunctNr:=T_Visu.T_CtrleAction.iFunction - 700;
				xActionProcMachine:=TRUE;
				tTimeOutAction:=T#0s;
		(* Stoppen vom Prozess welches über den Automat ausgelöst wurde *)
		799:		xProcMachineStop:=TRUE;
				tTimeOutAction:=T#0s;
		(* Save NovRAM without confirmation *)
		1001:	xAction_SaveNovRAM:=TRUE;
				tTimeOutAction:=T#10s;
		(* Erstmalige Kopiervorgang der Profile *)
		1002:	xAction_CopyProfileToProcess:=TRUE;
				tTimeOutAction:=T#60s;
		(* Laden eines ausgewählten Profil in den Prozessabbild *)
		1003:	xAction_LoadProfile:=TRUE;
				tTimeOutAction:=T#6s;
		(* Speichern eines ausgewählten Profils *)
		1004:	xAction_SaveProfile:=TRUE;
				tTimeOutAction:=T#6s;
		(* Löschen eines ausgewählten Profil *)
		1005:	xActionDeleteProfile:=TRUE;
				tTimeOutAction:=T#6s;
		(* change page from Taskbar *)
		10001..10999:	xSetNewPage:=TRUE;
					T_Visu.T_PlcParam.dwSetNewPage:=INT_TO_DWORD(T_Visu.T_CtrleAction.iFunction - 10000);
					tTimeOutAction:=T#3s;
		(* change page from Panel left Button *)
		11001..11999:	xSetParameterPage:=TRUE;
					T_Visu.T_PlcParam.dwSetNewPage:=INT_TO_DWORD(T_Visu.T_CtrleAction.iFunction - 11000);
					tTimeOutAction:=T#3s;
		ELSE
		(* function not implemented *)
			T_Visu.T_CtrleAction.xDone:=FALSE;
			T_Visu.T_CtrleAction.xNotReady:=FALSE;
			T_Visu.T_CtrleAction.xErr:=TRUE;
			T_Visu.T_CtrleAction.udiErrorID:=16#F000;
			(* exit FB *)
			RETURN;
		END_CASE
		(* Init. variable *)
		IF (T_ExchgParam.T_Visu.T_Message.iState = 401) THEN
			IF NOT(xSetNewPage) AND NOT(xSetPreviousPage) AND NOT(xPreviousPageVertical) AND
				NOT(xNextPageVertical) AND NOT(xResetErrorWarning) THEN
				(* Im Fehlerfall dürfen nur noch die Navigierung aktiviert sein und den Fehler zu Quittieren *)
					tTimeOutAction:=T#0s;
					T_Visu.T_CtrleAction.xDeleteVisuFunction:=TRUE;
					RETURN;
			END_IF;
		END_IF;
		T_Visu.T_CtrleAction.xDone:=FALSE;
		T_Visu.T_CtrleAction.xNotReady:=FALSE;
		T_Visu.T_CtrleAction.xErr:=FALSE;
		T_Visu.T_CtrleAction.udiErrorID:=0;
		iStepAction:=1;
		iStepActionNovRam:=1;
		iStepActionRef:=1;
		xStepActionDone:=FALSE;
		xBlockSetNovRamAction_End:=FALSE;	(* Mittels diesem Flag kann verhindert werden, dass die VisuFunktion für das speichern der Daten in den NovRam das EndFlag nicht gesetzt wird *)
		IF tTimeOutAction <> T#0s THEN TimerAction(IN:=FALSE); END_IF
		(* exit FB *)
		RETURN;
	END_IF;
(* Timer action *)
	IF tTimeOutAction <> T#0s THEN TimerAction(IN:=TRUE,PT:=tTimeOutAction); END_IF
	RisingEdgeTimeOut(CLK:=TimerAction.Q);
	IF RisingEdgeTimeOut.Q AND NOT(T_Visu.T_CtrleAction.xDone) AND NOT(T_Visu.T_CtrleAction.xErr) THEN
	(* Timeout action activ *)
		(* call confirmation message *)
		IF NOT(T_Visu.T_CtrleAction.xFunctionActive) THEN
			T_ExchgParam.T_Visu.T_Message.iState:=203;	(* Warnung: Ausführungszeit überschritten ! *)
			(* exit FB, do not continue the execution of action! *)
			T_Visu.T_CtrleAction.xDeleteVisuFunction:=TRUE;
			RETURN;
		END_IF;
	END_IF

(* Überprüfe für aufgerufene Visu Funktion ob die Energieversorgung eingeschaltet ist *)
	xCheckVisuFunctionPowerON:=FALSE;
	IF NOT(gT_SafetyStatus.xSetupOperateModeActive) THEN
		IF NOT(T_ExchgParam.T_SafetyCtrl.xNormalOperate_EnergyON)THEN
			xCheckVisuFunctionPowerON:=TRUE;
		END_IF;
	ELSE
		IF (gT_SafetyStatus.iSetupMode = 1) THEN
			IF NOT(T_ExchgParam.T_SafetyCtrl.xSetupOperateA_EnergyON)THEN
				xCheckVisuFunctionPowerON:=TRUE;
			END_IF;
		ELSIF (gT_SafetyStatus.iSetupMode = 2) THEN
			IF NOT(T_ExchgParam.T_SafetyCtrl.xSetupOperateB_EnergyON)THEN
				xCheckVisuFunctionPowerON:=TRUE;
			END_IF;
		END_IF;
	END_IF;
	IF xCheckVisuFunctionPowerON AND NOT(gxHardwareOFF) THEN
		xCheckVisuFunctionPowerON:=	xAxisStop OR xAxisStopAll OR xAxisTogglePower OR xAxisReset OR xZAxisMoveToToolChangePos OR xZAxisMoveToLoadPos;
		xCheckVisuFunctionPowerON:=	xCheckVisuFunctionPowerON OR xAxisMoveContinous OR xAxisMoveAbsolut OR xAxisMoveRelative;
		xCheckVisuFunctionPowerON:=	xCheckVisuFunctionPowerON OR xAxisTeachPosition OR xStationSetupAxisZFunction OR xStationSetupAxisZFunctionToolGuide;
		xCheckVisuFunctionPowerON:=	xCheckVisuFunctionPowerON OR xTmpStationSetupAxisZFunction OR xTmpStationSetupAxisZFunctionToolGuide;
		xCheckVisuFunctionPowerON:=	xCheckVisuFunctionPowerON OR xCylValveToggleOnOff OR xCylSetServoAnalogValue OR xCylPressurelessON OR xCylTorqueOnOff OR xCylTorqueOverloadOnOff;
		xCheckVisuFunctionPowerON:=	xCheckVisuFunctionPowerON OR xStationWorkFunction OR xSuspensionONOFF;
		xCheckVisuFunctionPowerON:=	xCheckVisuFunctionPowerON OR xStationToolCalibrateFunction OR xStationSpindleBurnInFunction;
		xCheckVisuFunctionPowerON:=	xCheckVisuFunctionPowerON OR xStationStop OR xStationStopWorkRight;
		xCheckVisuFunctionPowerON:=	xCheckVisuFunctionPowerON OR xActionProcStation OR xProcStationStop OR xActionProcMachine;
		xCheckVisuFunctionPowerON:=	xCheckVisuFunctionPowerON OR xTmpProcMachineStop;
		IF xCheckVisuFunctionPowerON THEN
			tTimeOutAction:=T#0s;
			TimerAction(IN:=FALSE);
			T_ExchgParam.T_Visu.T_Message.iState:=230;	(* Warnung: Zuerst die Energieversorgung einschalten ! *)
			T_Visu.T_CtrleAction.xDeleteVisuFunction:=TRUE;
			T_Visu.T_CtrleAction.xFunctionActive:=FALSE;
		END_IF;
	END_IF;

	IF (T_ExchgParam.T_Visu.T_Message.iState = 401) THEN
		IF NOT(xSetNewPage) AND NOT(xSetPreviousPage) AND NOT(xPreviousPageVertical) AND
		     NOT(xNextPageVertical) AND NOT(xResetErrorWarning) THEN
			(* Im Fehlerfall dürfen nur noch die Navigierung aktiviert sein und den Fehler zu Quittieren *)
			tTimeOutAction:=T#0s;
			T_Visu.T_CtrleAction.xDeleteVisuFunction:=TRUE;
			T_Visu.T_CtrleAction.xFunctionActive:=FALSE;
		END_IF;
	END_IF;

CtrlVisuFunctionDelete;
END_ACTION
ACTION CtrlVisuFunctionDelete:
(* Löschen aller Visu Funktionen *)
	IF T_Visu.T_CtrleAction.xDeleteVisuFunction THEN
		T_Visu.T_CtrleAction.xDeleteVisuFunction:=FALSE;
		T_Visu.T_CtrleAction.xExecute:=FALSE;
		T_Visu.T_CtrleAction.xDone:=TRUE;
		T_Visu.T_CtrleAction.xNotReady:=FALSE;
		T_Visu.T_CtrleAction.xErr:=FALSE;
		T_Visu.T_CtrleAction.udiErrorID:=16#0;
		T_StartUp.T_State.xBlockChangeMovementVisu:=FALSE;
		xSetNewPage:=FALSE;
		xSetParameterPage:=FALSE;
		xSetPreviousPage:=FALSE;
		xPreviousPageVertical:=FALSE;
		xNextPageVertical:=FALSE;
		xDeleteErrorList:=FALSE;
		xResetErrorWarning:=FALSE;
		xLampTestOnOff:=FALSE;
		xLampTestBlinkOnOff:=FALSE;
		xLampTestActive:=FALSE;
		xOpenMessageWindow:=FALSE;
		xMachineDoorUpGuardControlTogOnOff:=FALSE;
		xChangeOperatorPassword:=FALSE;
		xProcessStation1ResetToolChange:=FALSE;
		xOnlineChange_TorqueLevelHCMore:=FALSE;
		xOnlineChange_TorqueLevelHCLess:=FALSE;
		xOnlineChange_DeflectionForceMore:=FALSE;
		xOnlineChange_DeflectionForceLess:=FALSE;
		xOnlineChange_Z_ForwardSpeedMore:=FALSE;
		xOnlineChange_Z_ForwardSpeedLess:=FALSE;
		xOnlineChange_Z_BackwardSpeedMore:=FALSE;
		xOnlineChange_Z_BackwardSpeedLess:=FALSE;
		xOnlineChange_Z_BackwardOffsetMore:=FALSE;
		xOnlineChange_Z_BackwardOffsetLess:=FALSE;
		xOnlineChange_S_WorkSpeedMore:=FALSE;
		xOnlineChange_S_WorkSpeedLess:=FALSE;
		xTorqueOffsetMinus:=FALSE;
		xTorqueOffsetPlus:=FALSE;
		xSaveTorqueScale:=FALSE;
		xSaveTorquePosition:=FALSE;
		xSelectConfigPosition_1:=FALSE;
		xSelectConfigPosition_2:=FALSE;
		xSelectConfigPosition_3:=FALSE;
		xSelectConfigPosition_4:=FALSE;
		xSaveConfigPosition:=FALSE;
		xConfigPosOnOff:=FALSE;
		xSpindelCalibrationONOFF:=FALSE;
		xStationToolCalibrateFunction:=FALSE;
		xStationSpindleBurnInFunction:=FALSE;
		xDeleteProcessState:=FALSE;
		xEndlessProcessOnOff:=FALSE;
		xCentringONOFF:=FALSE;
		xOnlyCentringONOFF:=FALSE;
		xSuspensionONOFF:=FALSE;
		xSetupPotentiometer:=FALSE;
		xZAxisMoveToToolChangePos:=FALSE;
		xZAxisMoveToLoadPos:=FALSE;
		xZSaveEndPosCalc:=FALSE;
		xSelectZInkWorkInfo:=FALSE;
		xSelectZInkCentringInfo:=FALSE;
		xAxisStop:=FALSE;
		xAxisStopAll:=FALSE;
		xAxisTogglePower:=FALSE;
		xAxisReset:=FALSE;
		xAxisMoveContinous:=FALSE;
		xAxisMoveAbsolut:=FALSE;
		xAxisMoveRelative:=FALSE;
		xAxisTeachPosition:=FALSE;
		xResetRockerValue:=FALSE;
		xCylValveToggleOnOff:=FALSE;
		xCylTorqueOnOff:=FALSE;
		xCylTorqueOverloadOnOff:=FALSE;
		xCylSetServoAnalogValue:=FALSE;
		xCylPressurelessON:=FALSE;
		xStationWorkFunction:=FALSE;
		xStationStop:=FALSE;
		xStationStopWorkRight:=FALSE;
		xActionProcStation:=FALSE;
		xProcStationStop:=FALSE;
		xActionProcMachine:=FALSE;
		xProcMachineStop:=FALSE;
		xTmpProcMachineStop:=FALSE;
		xAction_SaveNovRAM:=FALSE;
		xAction_CopyProfileToProcess:=FALSE;
		xAction_LoadProfile:=FALSE;
		xAction_SaveProfile:=FALSE;
		xActionDeleteProfile:=FALSE;
		xStationSetupAxisZFunction:=FALSE;
		xTmpStationSetupAxisZFunction:=FALSE;
		xStationSetupAxisZFunctionToolGuide:=FALSE;
		xTmpStationSetupAxisZFunctionToolGuide:=FALSE;
		xRegulatorOverlaySave:=FALSE;
		xRegulatorType1:=FALSE;
		xRegulatorType2:=FALSE;
		xRegulatorType3:=FALSE;
	END_IF;
END_ACTION
ACTION InitQVIS:
(* determin if qvis activ *)
	IF xQvisActiv THEN
		(* timer time off  *)
		TimerQVis(IN:=TRUE,PT:=T#2s);
		IF dwInCount_QVisCmd = T_CtrleQVis.dwInCount THEN
			(* Init. command *)
			T_CtrleQVis.dwInCommand:=1;
			T_CtrleQVis.dwInQVisCtrlAddress:=ADR(T_CtrleQVis);
			T_CtrleQVis.dwInParameterAddress:=ADR(T_Visu.T_PlcParam.dwSetNewPage);
			(* start command *)
			T_CtrleQVis.dwInCount:=T_CtrleQVis.dwInCount+1;
			(* Activ Timer *)
			TimerQVis(IN:=FALSE);
		ELSE
			IF T_CtrleQVis.dwInCount = T_CtrleQVis.dwOutCount THEN
			(* command done *)
				IF T_CtrleQVis.diOutStatus = 0 THEN
				(* command done without error *)
					xQvisActiv:=FALSE;
					T_Visu.T_CtrleVisu.xQvis:=TRUE;
					T_Visu.T_PlcParam.dwActualPage:=T_Visu.T_PlcParam.dwSetNewPage;
				END_IF
			ELSE
			(* test time off, restart command *)
				IF TimerQVis.Q THEN
					dwInCount_QVisCmd:=T_CtrleQVis.dwInCount;
				END_IF
			END_IF
		END_IF
	END_IF

(* Überprüfe ob die QVisRuntime noch am leben ist *)
IF T_StartUp.T_State.xPLCReady THEN
	TONWaitCheckQVis(IN:=TRUE,PT:=T#5s);
	IF TONWaitCheckQVis.Q THEN
		CASE iStepCheckQVis OF
		1:	IF NOT(T_Visu.T_CtrleVisu.xExecute) AND T_Visu.T_CtrleVisu.xDone AND NOT(xChangePage) THEN	(* Abwarten bis Visu Ressource frei steht *)
				xBlockChangeVisuPage:=TRUE;
				IF (T_CtrleQVis.dwInCount > 4294967295) THEN
					T_CtrleQVis.dwInCount:=0;
				END_IF;
				T_CtrleQVis.dwInCount:=T_CtrleQVis.dwInCount + 1;
				iStepCheckQVis:=iStepCheckQVis + 1;
				TONWaitLiftTime(IN:=FALSE);
			END_IF;
		2:	TONWaitLiftTime(IN:=TRUE,PT:=T#2000ms);
			IF TONWaitLiftTime.Q THEN
				TONWaitLiftTime(IN:=FALSE);
				xBlockChangeVisuPage:=FALSE;
				T_StartUp.T_Ctrle.iFunction:=5;	(* Booting Funktion *)
				T_StartUp.T_Ctrle.xExecute:=TRUE;
				T_Visu.T_CtrleVisu.xReset:=TRUE;
				T_Visu.T_CtrleVisu.xQvis:=FALSE;
				xQvisActiv:=TRUE;
			END_IF;
			IF T_CtrleQVis.dwInCount = T_CtrleQVis.dwOutCount THEN
				TONWaitCheckQVis(IN:=FALSE);
				TONWaitLiftTime(IN:=FALSE);
				xBlockChangeVisuPage:=FALSE;
			END_IF;
		END_CASE;
	ELSE
		iStepCheckQVis:=1;
	END_IF;
ELSE
	iStepCheckQVis:=1;
	TONWaitCheckQVis(IN:=FALSE);
	TONWaitLiftTime(IN:=FALSE);
	xBlockChangeVisuPage:=FALSE;
END_IF;
END_ACTION
ACTION InitSavePages:
dwSaveActualPageTask[0,1]:=10;
dwSaveActualPageTask[0,2]:=20;
dwSaveActualPageTask[0,3]:=30;
dwSaveActualPageTask[0,4]:=40;
dwSaveActualPageTask[0,5]:=50;
dwSaveActualPageTask[0,6]:=60;

dwSaveActualPageTask[1,1]:=110;
dwSaveActualPageTask[1,2]:=120;
dwSaveActualPageTask[1,3]:=130;
dwSaveActualPageTask[1,4]:=140;
dwSaveActualPageTask[1,5]:=150;
dwSaveActualPageTask[1,6]:=160;

dwSaveActualPageTask[2,1]:=210;
dwSaveActualPageTask[2,2]:=220;
dwSaveActualPageTask[2,3]:=230;
dwSaveActualPageTask[2,4]:=240;
dwSaveActualPageTask[2,5]:=250;
dwSaveActualPageTask[2,6]:=260;

dwSaveActualPageTask[3,1]:=310;
dwSaveActualPageTask[3,2]:=320;
dwSaveActualPageTask[3,3]:=330;
dwSaveActualPageTask[3,4]:=340;
dwSaveActualPageTask[3,5]:=350;
dwSaveActualPageTask[3,6]:=360;
END_ACTION
ACTION MaskFunctionButton:
	IF (T_Visu.T_PlcParam.dwActualPage = gT_PageNumber.iAutoMode_UserLevel) AND (T_ExchgParam.T_Visu.T_Level.iActLevel = 1) THEN
		(* Wenn der OperatorLevel Aktiv ist, dann muss die F1 Funktionstaste zur Verfügung gestellt werden um den Passwort ändern zu können *)
		IF TProcess.T_Ctrle.xDone AND NOT(TProcess.T_Ctrle.xError) THEN
			wForceMaskFunctionPanel:=16#1;
		END_IF;
	END_IF;

	CASE T_Visu.T_PlcParam.dwActualPage OF

	gT_PageNumber.iAutoMode_PartQuality:
		IF (T_ExchgParam.T_Visu.T_Level.iActLevel >= 1) THEN
			wForceMaskFunctionPanel:=16#1;
		END_IF;

	gT_PageNumber.iAutoMode_SafetyCheck:
		IF NOT(TProcess.T_Ctrle.xDone) THEN
			(* Wenn mindestens ein Prozess Aktiv ist von einer Arbeitsstation dann darf unabhängig der ausgewählten Arbeitsstation die Türzuhaltung mittels der F1 Taste nicht geöffnet werden *)
			wForceMaskFunctionPanel:=2#1000000;	(* F1 unterdrücken, dazu wird F7 freigegeben (F7 gibt es auf dieser Seite nicht) weil sonst mit Null die Maske nicht überschrieben wird *)
		END_IF;

	gT_PageNumber.iAutoMode_ToolChange:
		IF NOT(T_NovRam.T_Parameter.T_StationWork[1].T_StProcess.xPositionEndProcIncOnOff) AND (T_ExchgParam.T_StationCommon.bSelectShowIncValue = 0) THEN
			wForceMaskFunctionPanel:=16#1F;
		END_IF;
		IF NOT(T_NovRam.T_Parameter.T_StationWork[1].T_StProcess.xCentringEndProcIncOnOff) AND (T_ExchgParam.T_StationCommon.bSelectShowIncValue = 1) THEN
			wForceMaskFunctionPanel:=16#1F;
		END_IF;

	gT_PageNumber.iWorkStation_Axis1:
		CASE T_ExchgParam.T_TeachIn.iSetup_AxisSel OF
		gciAxisZ_St1:			(* Z Achse: *)
			wForceMaskFunctionPanel:=16#33;
			aiForceRTrigActionFunctionPanel[1]:=203;
			aiForceRTrigActionFunctionPanel[2]:=204;
			aiForceRTrigActionFunctionPanel[3]:=0;
			aiForceRTrigActionFunctionPanel[4]:=0;
			aiForceRTrigActionFunctionPanel[5]:=185;	(* KonfigPos EIN/AUS *)
			aiForceRTrigActionFunctionPanel[6]:=214;
		gciAxisS_St1:			(* Maxon Spindel: *)
			wForceMaskFunctionPanel:=16#3B;
			aiForceRTrigActionFunctionPanel[1]:=203;
			aiForceRTrigActionFunctionPanel[2]:=204;
			aiForceRTrigActionFunctionPanel[3]:=0;
			aiForceRTrigActionFunctionPanel[4]:=121;		(* OnlineChange Parameter Zylinder ToolTorque Drehmoment Schwellwert 1 Start Position - *)
			aiForceRTrigActionFunctionPanel[5]:=120;		(* OnlineChange Parameter Zylinder ToolTorque Drehmoment Schwellwert 1 Start Position + *)
			aiForceRTrigActionFunctionPanel[6]:=230;		(* Löschen der berechnete Wert für Wippe des Drehmoment Detection *)
		3:					(* Beckhoff Spindel: *)
			wForceMaskFunctionPanel:=16#3;
			aiForceRTrigActionFunctionPanel[1]:=203;
			aiForceRTrigActionFunctionPanel[2]:=204;
			aiForceRTrigActionFunctionPanel[3]:=0;
			aiForceRTrigActionFunctionPanel[4]:=0;
			aiForceRTrigActionFunctionPanel[5]:=0;
			aiForceRTrigActionFunctionPanel[6]:=0;
		END_CASE;

	gT_PageNumber.iHandMode_OnlineChange:
		wForceMaskFunctionPanel:=16#FFF;
		aiForceRTrigActionFunctionPanel[1]:=120;		(* OnlineChange Parameter Zylinder ToolTorque Drehmoment Schwellwert HC + *)
		aiForceRTrigActionFunctionPanel[2]:=126;		(* OnlineChange Parameter Zylinder ToolDeflection Auslenkkraft + *)
		aiForceRTrigActionFunctionPanel[3]:=128;		(* OnlineChange Parameter Z Achse Bearbeitungsgeschwindigkeit vorwärts + *)
		aiForceRTrigActionFunctionPanel[4]:=132;		(* OnlineChange Parameter Z Achse rückwärts Offset + *)
		aiForceRTrigActionFunctionPanel[5]:=130;		(* OnlineChange Parameter Z Achse Bearbeitungsgeschwindigkeit rückwärts + *)
		aiForceRTrigActionFunctionPanel[6]:=134;		(* OnlineChange Parameter S Achse Bearbeitungsgeschwindigkeit + *)
		aiForceRTrigActionFunctionPanel[7]:=121;		(* OnlineChange Parameter Zylinder ToolTorque Drehmoment Schwellwert HC - *)
		aiForceRTrigActionFunctionPanel[8]:=127;		(* OnlineChange Parameter Zylinder ToolDeflection Auslenkkraft - *)
		aiForceRTrigActionFunctionPanel[9]:=129;		(* OnlineChange Parameter Z Achse Bearbeitungsgeschwindigkeit vorwärts - *)
		aiForceRTrigActionFunctionPanel[10]:=133;		(* OnlineChange Parameter Z Achse rückwärts Offset - *)
		aiForceRTrigActionFunctionPanel[11]:=131;		(* OnlineChange Parameter Z Achse Bearbeitungsgeschwindigkeit rückwärts - *)
		aiForceRTrigActionFunctionPanel[12]:=135;		(* OnlineChange Parameter S Achse Bearbeitungsgeschwindigkeit + *)

	gT_PageNumber.iHandMode_Setup1:
		IF TProcess.T_Ctrle.xDone AND NOT(TProcess.T_Ctrle.xError) THEN
			IF xSetupPotentiometer THEN
				IF (iStepAction = 20) THEN
					wForceMaskFunctionPanel:=16#20;
				END_IF;
			ELSE
				wForceMaskFunctionPanel:=16#1;
			END_IF;
		ELSE
			wForceMaskFunctionPanel:=16#1000;
		END_IF;

	gT_PageNumber.iWorkStation_Setup4:
		CASE T_ExchgParam.bToolSpindleActive OF
		1:	(* Maxon Spindel *)
			wForceMaskFunctionPanel:=16#3F;
			aiForceRTrigActionFunctionPanel[1]:=171;	(* Torque Offset - *)
			aiForceRTrigActionFunctionPanel[2]:=172;	(* Torque Offset - *)
			aiForceRTrigActionFunctionPanel[3]:=303;	(* Zyl WzDrehmoment EIN/AUS *)
			aiForceRTrigActionFunctionPanel[4]:=304;	(* Zyl WzDrehmomentÜberlast EIN/AUS *)
			aiForceRTrigActionFunctionPanel[5]:=173;	(* Save Torque Scale *)
			aiForceRTrigActionFunctionPanel[6]:=174;	(* Save Torque Position *)
		2,3:	(* Beckhoff Spindel *)
			wForceMaskFunctionPanel:=16#F000;
			aiForceRTrigActionFunctionPanel[1]:=0;
			aiForceRTrigActionFunctionPanel[2]:=0;
			aiForceRTrigActionFunctionPanel[3]:=0;
			aiForceRTrigActionFunctionPanel[4]:=0;
			aiForceRTrigActionFunctionPanel[5]:=0;
			aiForceRTrigActionFunctionPanel[6]:=0;
		END_CASE;


	END_CASE;
END_ACTION
ACTION MaskRightButton:
	IF (T_Visu.T_PlcParam.dwActualPage = gT_PageNumber.iWorkStation_Axis1) THEN
		CASE T_ExchgParam.T_TeachIn.iSetup_AxisSel OF
		gciAxisZ_St1:		wForceMaskBtPanelRight:=16#60;
		gciAxisS_St1,3:	wForceMaskBtPanelRight:=16#0;
		END_CASE;
	END_IF;
END_ACTION
ACTION Monitor_ActuatorState:
(*******************************************************************************************************************************************************************************************)
(*************************************************			                                   Zylinder Zustand abfragen                                                     ******************************************)
(*******************************************************************************************************************************************************************************************)
(* 01 WzAuslenkung St1 *)
	T_ExchgParam.T_Cylinder.arStat[1].xOff:=	FALSE;
	T_ExchgParam.T_Cylinder.arStat[1].xOn:=	TStation_Work_St1.THWWorkStation.TCylToolDeflection.T_CtrleCyl.T_Analog.xActiv;
	T_ExchgParam.T_Cylinder.arStat[1].bStat:=	bFct_SetCylStat(	TStation_Work_St1.THWWorkStation.TCylToolDeflection.T_CtrleCyl.xStatePosOff,
														 		TStation_Work_St1.THWWorkStation.TCylToolDeflection.T_CtrleCyl.xStatePosOn,
											 					T_ExchgParam.T_Cylinder.arStat[1].bStat);
(* 02 Servoventil für Drehmomentüberwachung HC *)
	T_ExchgParam.T_Cylinder.arStat[2].xOff:=	FALSE;
	T_ExchgParam.T_Cylinder.arStat[2].xOn:=	TStation_Work_St1.THWWorkStation.TCylToolTorqueHC.T_CtrleCyl.T_Analog.xActiv;
	T_ExchgParam.T_Cylinder.arStat[2].bStat:=	bFct_SetCylStat(	TStation_Work_St1.THWWorkStation.TCylToolTorqueHC.T_CtrleCyl.xStatePosOff,
														 		TStation_Work_St1.THWWorkStation.TCylToolTorqueHC.T_CtrleCyl.xStatePosOn,
											 					T_ExchgParam.T_Cylinder.arStat[2].bStat);
(* 03 Servoventil für Drehmomentüberwachung Überlast *)
	T_ExchgParam.T_Cylinder.arStat[3].xOff:=	FALSE;
	T_ExchgParam.T_Cylinder.arStat[3].xOn:=	TStation_Work_St1.THWWorkStation.TCylToolTorqueOverload.T_CtrleCyl.T_Analog.xActiv;
	T_ExchgParam.T_Cylinder.arStat[3].bStat:=	bFct_SetCylStat(	TStation_Work_St1.THWWorkStation.TCylToolTorqueOverload.T_CtrleCyl.xStatePosOff,
														 		TStation_Work_St1.THWWorkStation.TCylToolTorqueOverload.T_CtrleCyl.xStatePosOn,
											 					T_ExchgParam.T_Cylinder.arStat[3].bStat);
(* 04 Bremse Z Achse St1 *)
	T_ExchgParam.T_Cylinder.arStat[4].xOff:=	TStation_Work_St1.THWWorkStation.TCylBrakeReleaseZAxis.T_CtrleCyl.T_Standard.xActivOff;
	T_ExchgParam.T_Cylinder.arStat[4].xOn:=	TStation_Work_St1.THWWorkStation.TCylBrakeReleaseZAxis.T_CtrleCyl.T_Standard.xActivOn;
	T_ExchgParam.T_Cylinder.arStat[4].bStat:=	bFct_SetCylStat(	TStation_Work_St1.THWWorkStation.TCylBrakeReleaseZAxis.T_CtrleCyl.xStatePosOff,
														 		TStation_Work_St1.THWWorkStation.TCylBrakeReleaseZAxis.T_CtrleCyl.xStatePosOn,
											 					T_ExchgParam.T_Cylinder.arStat[4].bStat);
(* 05 Werkstück Spannung *)
	T_ExchgParam.T_Cylinder.arStat[5].xOff:=	FALSE;
	T_ExchgParam.T_Cylinder.arStat[5].xOn:=	TStation_Work_St1.THWWorkStation.TCylWorkpieceClamp.T_CtrleCyl.T_Standard.xActivOn;
	T_ExchgParam.T_Cylinder.arStat[5].bStat:=	bFct_SetCylStat(	TStation_Work_St1.THWWorkStation.TCylWorkpieceClamp.T_CtrleCyl.xStatePosOff,
														 		TStation_Work_St1.THWWorkStation.TCylWorkpieceClamp.T_CtrleCyl.xStatePosOn,
											 					T_ExchgParam.T_Cylinder.arStat[5].bStat);
(* 06 Ventil Luft Tisch *)
	T_ExchgParam.T_Cylinder.arStat[6].xOff:=	TStation_Work_St1.THWWorkStation.TValveAirTable.T_CtrleCyl.T_Standard.xActivOff;
	T_ExchgParam.T_Cylinder.arStat[6].xOn:=	TStation_Work_St1.THWWorkStation.TValveAirTable.T_CtrleCyl.T_Standard.xActivOn;
	T_ExchgParam.T_Cylinder.arStat[6].bStat:=	bFct_SetCylStat(	TStation_Work_St1.THWWorkStation.TValveAirTable.T_CtrleCyl.xStatePosOff,
														 		TStation_Work_St1.THWWorkStation.TValveAirTable.T_CtrleCyl.xStatePosOn,
											 					T_ExchgParam.T_Cylinder.arStat[6].bStat);
(* 07 Ventil Vakuum Tisch *)
	T_ExchgParam.T_Cylinder.arStat[7].xOff:=	TStation_Work_St1.THWWorkStation.TValveVacuumTable.T_CtrleCyl.T_Standard.xActivOff;
	T_ExchgParam.T_Cylinder.arStat[7].xOn:=	TStation_Work_St1.THWWorkStation.TValveVacuumTable.T_CtrleCyl.T_Standard.xActivOn;
	T_ExchgParam.T_Cylinder.arStat[7].bStat:=	bFct_SetCylStat(	TStation_Work_St1.THWWorkStation.TValveVacuumTable.T_CtrleCyl.xStatePosOff,
														 		TStation_Work_St1.THWWorkStation.TValveVacuumTable.T_CtrleCyl.xStatePosOn,
											 					T_ExchgParam.T_Cylinder.arStat[7].bStat);
(*******************************************************************************************************************************************************************************************)
(*************************************************			                                   Achsen Zustand abfragen                                                      ******************************************)
(*******************************************************************************************************************************************************************************************)
(*  Reihenfolge Achsen Anwahl: *)
(*1:Achse Z,*)
T_ExchgParam.T_TeachIn.arAxis[gciAxisZ_St1].bActState	:=
		bFct_SetAxisStat(	TStation_Work_St1.THWWorkStation.TAxisZ.T_CtrleSingle.xPower,
							TStation_Work_St1.THWWorkStation.TAxisZ.T_CtrleSingle.xRef,
							NOT TStation_Work_St1.THWWorkStation.TAxisZ.T_CtrleSingle.xNotMoving ,
							TStation_Work_St1.THWWorkStation.TAxisZ.T_CtrleSingle.xErr,
							TStation_Work_St1.THWWorkStation.TAxisZ.T_CtrleSingle.xStateHWLimitNeg,
							TStation_Work_St1.THWWorkStation.TAxisZ.T_CtrleSingle.xStateHWLimitPos,
							T_ExchgParam.T_TeachIn.arAxis[gciAxisZ_St1].bActState);
T_ExchgParam.T_TeachIn.arAxis[gciAxisZ_St1].rActPos		:=TStation_Work_St1.THWWorkStation.TAxisZ.T_LiveValue.lrActualPosition;
T_ExchgParam.T_TeachIn.arAxis[gciAxisZ_St1].rActSpeed	:=TStation_Work_St1.THWWorkStation.TAxisZ.T_LiveValue.lrActualVelocity;
(*5:Achse S,*)
T_ExchgParam.T_TeachIn.arAxis[gciAxisS_St1].bActState	:=
		bFct_SetAxisStat(	TStation_Work_St1.THWWorkStation.TAxisS.T_CtrleSingle.xPower,
							TStation_Work_St1.THWWorkStation.TAxisS.T_CtrleSingle.xRef,
							NOT TStation_Work_St1.THWWorkStation.TAxisS.T_CtrleSingle.xNotMoving ,
							TStation_Work_St1.THWWorkStation.TAxisS.T_CtrleSingle.xErr,
							TStation_Work_St1.THWWorkStation.TAxisS.T_CtrleSingle.xStateHWLimitNeg,
							TStation_Work_St1.THWWorkStation.TAxisS.T_CtrleSingle.xStateHWLimitPos,
							T_ExchgParam.T_TeachIn.arAxis[gciAxisS_St1].bActState);
T_ExchgParam.T_TeachIn.arAxis[gciAxisS_St1].rActPos		:=TStation_Work_St1.THWWorkStation.TAxisS.T_LiveValue.lrActualPosition;
T_ExchgParam.T_TeachIn.arAxis[gciAxisS_St1].rActSpeed	:=TStation_Work_St1.THWWorkStation.TAxisS.T_LiveValue.lrActualVelocity;
CASE T_ExchgParam.T_TeachIn.iSetup_AxisSel OF
gciAxisZ_St1:		T_ExchgParam.T_TeachIn.rTeachSelStep:=T_ExchgParam.T_TeachIn.arTeachSelStep[gciAxisZ_St1];
				T_ExchgParam.T_TeachIn.rTeachSelVel:=T_ExchgParam.T_TeachIn.arTeachSelVel[gciAxisZ_St1];
gciAxisS_St1,3:	T_ExchgParam.T_TeachIn.rTeachSelStep:=T_ExchgParam.T_TeachIn.arTeachSelStep[gciAxisS_St1];
				T_ExchgParam.T_TeachIn.rTeachSelVel:=T_ExchgParam.T_TeachIn.arTeachSelVel[gciAxisS_St1];
END_CASE;
(*++++++++++++++++Teach Positions WorkStation++++++++++++++++
POSITIONS FOR  Z Axis!
0:=< Fahre zu man. Pos. >
1:=< Z LadePos >
2:=< Z Bearb StartPos >
3:=< Z Bearb EndPos >
4:=< Z WzWechsel Pos >
5:=< Z Mech EndPos > *)
(*Call Function selected Teach Pos to HMI *)
FBTeachPosToHMI(	iAxisNr:= 1,
					iSelectPos:= T_ExchgParam.T_TeachIn.arAxis[gciAxisZ_St1].iTeachSelPos,
					rSetPos:= T_ExchgParam.T_TeachIn.arAxis[gciAxisZ_St1].rSetPos,
					TeachPosWork:= T_NovRam.T_Parameter.T_StationWork[gciStationSt1].T_StProcess);
T_ExchgParam.T_TeachIn.arAxis[gciAxisZ_St1].rTeachPosStored:=FBTeachPosToHMI.rPosition;
END_ACTION
ACTION Monitor_FctButton_Led:
(* Aktivierungsanzeige der Funktionstasten *)
wTmp:=0;
CASE T_Visu.T_PlcParam.dwActualPage OF
	gT_PageNumber.iAutoMode_Process:
		(* F1-->Endlos Prozess EIN/AUS *)
		IF T_NovRAM.T_Parameter.T_Machine.xEndlessProcessActive THEN wTmp:=wTmp OR 16#1; END_IF;
		(* F2-->Zentrieren EIN/AUS *)
		IF gxCentringActive THEN wTmp:=wTmp OR 16#2; END_IF;
		(* F3-->NurZentrieren EIN/AUS *)
		IF gxOnlyCentringActive THEN wTmp:=wTmp OR 16#4; END_IF;
		(* F4-->Suspension EIN/AUS *)
		IF NOT(TStation_Work_St1.THWWorkStation.TAxisBubbler.T_CtrleDCAxis.xNotMoving) OR NOT(TStation_Work_St1.THWWorkStation.TAxisFeedPump.T_CtrleDCAxis.xNotMoving) THEN wTmp:=wTmp OR 16#8; END_IF;
		(* F5-->ZylWPUnfix EIN/AUS *)
		IF QxCylWPUnfix_St1 THEN wTmp:=wTmp OR 16#10; END_IF;
	gT_PageNumber.iAutoMode_Referencing:
		(* F1-->Spindelkalibrierung EIN/AUS St1 *)
		IF  gxSpindelCalibrationONOFF_St1 THEN
			wTmp:=wTmp OR 16#1;
		END_IF;
	gT_PageNumber.iAutoMode_ToolChange:
		(* F1-->Station 1 WzWechsel Zähler zurücksetzen *)
		IF xProcessStation1ResetToolChange THEN wTmp:=wTmp OR 16#1; END_IF
		(* F2-->Z WzWechselPos *)
		IF xZAxisMoveToToolChangePos THEN wTmp:=wTmp OR 16#2; END_IF
		(* F3-->Z LadePos *)
		IF xZAxisMoveToLoadPos THEN wTmp:=wTmp OR 16#4; END_IF
		(* F4-->Auswahl Anzeige Ink Werte Bearbeitung *)
		IF (T_ExchgParam.T_StationCommon.bSelectShowIncValue = 0) THEN wTmp:=wTmp OR 16#8; END_IF;
		(* F5-->Auswahl Anzeige Ink Werte Bearbeitung *)
		IF (T_ExchgParam.T_StationCommon.bSelectShowIncValue = 1) THEN wTmp:=wTmp OR 16#10; END_IF;
		(* F6-->Speichern Z EndPos Berechnet *)
		IF xZSaveEndPosCalc THEN wTmp:=wTmp OR 16#20; END_IF;
	gT_PageNumber.iAutoMode_SafetyCheck:
		(* F1-->Türzuhaltung *)
		IF QxCabinDoorLock THEN wTmp:=wTmp OR 16#1; END_IF

	gT_PageNumber.iHandMode_RegulatorPara:
		(* F1-->Konv.Regler *)
		IF (T_NovRAM.T_Parameter.T_StationWork[1].T_StProcess.iWorkControlType <= 1) THEN wTmp:=wTmp OR 16#1; END_IF
		(* F2-->Adapt.Vorschub Regler *)
		IF (T_NovRAM.T_Parameter.T_StationWork[1].T_StProcess.iWorkControlType = 2) THEN wTmp:=wTmp OR 16#2; END_IF
		(* F1-->Konv.PD Regler *)
		IF (T_NovRAM.T_Parameter.T_StationWork[1].T_StProcess.iWorkControlType = 3) THEN wTmp:=wTmp OR 16#4; END_IF

	gT_PageNumber.iHandMode_ConfigPosition:
		(* F1-->Position Führungsrohr *)
		IF (T_ExchgParam.T_StationCommon.iSelectConfigPosition = 1) THEN wTmp:=wTmp OR 16#1; END_IF
		(* F2-->Abstand Führungsrohr *)
		IF (T_ExchgParam.T_StationCommon.iSelectConfigPosition = 2) THEN wTmp:=wTmp OR 16#2; END_IF
		(* F3-->Werkzeug *)
		IF (T_ExchgParam.T_StationCommon.iSelectConfigPosition = 3) THEN wTmp:=wTmp OR 16#4; END_IF
		(* F4-->Führungsrohr Einsatz *)
		IF (T_ExchgParam.T_StationCommon.iSelectConfigPosition = 4) THEN wTmp:=wTmp OR 16#8; END_IF
		(* F5-->KonfigPos EIN/AUS *)
		IF T_NovRam.T_Parameter.T_StationWork[1].T_StProcess.xConfigActive THEN wTmp:=wTmp OR 16#10; END_IF
	gT_PageNumber.iWorkStation_Axis1:
		(* F1-->Zustand Achsenstrom ON/OFF *)
		IF ptrTCommonAxis^.T_CtrleSingle.xPower THEN wTmp:=wTmp OR 16#1; END_IF;
		(* F2-->Achse ist am resetten *)
		IF  (ptrTCommonAxis^.T_CtrleSingle.iFunction = 1) AND NOT( ptrTCommonAxis^.T_CtrleSingle.xDone) AND NOT( ptrTCommonAxis^.T_CtrleSingle.xErr) THEN
			wTmp:=wTmp OR 16#2;
		END_IF;
		IF (ptrTCommonAxis^.T_Config_Gen.iTyp = 1) THEN
			(* F5-->KonfigPos EIN/AUS *)
			IF T_NovRam.T_Parameter.T_StationWork[1].T_StProcess.xConfigActive THEN wTmp:=wTmp OR 16#10; END_IF
			(* F6-->Speichervorgang aktiv *)
			IF xAxisTeachPosition THEN wTmp:=wTmp OR 16#20; END_IF;
		END_IF;
	gT_PageNumber.iWorkStation_Setup4:
		(* F3-->Zustand Zyl Drehmoment *)
		IF TStation_Work_St1.THWWorkStation.TCylToolTorqueHC.T_CtrleCyl.T_Analog.xActiv THEN wTmp:=wTmp OR 16#4; END_IF;
		(* F4-->Zustand Zyl Drehmoment Überlast *)
		IF TStation_Work_St1.THWWorkStation.TCylToolTorqueOverload.T_CtrleCyl.T_Analog.xActiv THEN wTmp:=wTmp OR 16#8; END_IF;
END_CASE;
T_ExchgParam.T_BtFunctionPanel.wState:=wTmp;
END_ACTION
ACTION Monitor_Function:
IF (T_Visu.T_PlcParam.dwActualPage = gT_PageNumber.iHandMode_Setup1) THEN
(* Setup Potentiometer *)
	T_ExchgParam.T_FunctionCommon.adiPotentiometerValue:=
										T_NovRam.T_Parameter.T_Machine.adiPotentiometerValue;
	T_ExchgParam.T_FunctionCommon.adiPotentiometerValue[11]:=
										T_NovRam.T_Parameter.T_Machine.adiPotentiometerValue[11]:=
										IiASpeedServoDrive;
END_IF;
END_ACTION
ACTION Monitor_Station:
(* Monitoring von Station 1-->Bearbeitungsstation MicroHead *)
IF (TStation_Work_St1.TControl.diErrorNr <> 0) THEN
	T_ExchgParam.T_Station1.diErrorNr:=TStation_Work_St1.TControl.diErrorNr;
ELSE
	T_ExchgParam.T_Station1.diErrorNr:=0;
END_IF;
T_ExchgParam.T_Station1.iProfile:=T_NovRam.T_Parameter.T_StationWork[gciStationSt1].T_InfoProcess.iProfile;
T_ExchgParam.T_Station1.sProfileName:=T_NovRam.T_Parameter.T_StationWork[gciStationSt1].T_InfoProcess.sProfileName;
T_ExchgParam.T_StationCommon.T_Param_Machine.T_ParamAutomat.tActualActiveTime_St1:=T_NovRAM.T_Parameter.T_Machine.T_ParamAutomat.tActualActiveTime_St1;
T_ExchgParam.T_StationCommon.T_Param_Machine.T_ParamAutomat.iActualActiveTime_St1:=T_NovRAM.T_Parameter.T_Machine.T_ParamAutomat.iActualActiveTime_St1;
T_ExchgParam.T_Station1.xExist:=TRUE;
T_ExchgParam.T_Station1.xActiv:=TRUE;
T_ExchgParam.T_Station1.wState:=16#0;
IF TStation_Work_St1.TControl.xEnable AND TStation_Work_St1.TControl.xRdy AND TStation_Work_St1.TControl.xReferenced THEN
	T_ExchgParam.T_Station1.wState:=T_ExchgParam.T_Station1.wState OR 16#1;		(* Maschine ist Referenziert *)
ELSE
	T_ExchgParam.T_Station1.wState:=T_ExchgParam.T_Station1.wState AND 16#FE;
END_IF;
IF (NOT(TStation_Work_St1.TControl.xDone) AND NOT(TStation_Work_St1.TControl.xError)) THEN
	T_ExchgParam.T_Station1.wState:=T_ExchgParam.T_Station1.wState OR 16#2;		(* Stationsfunktion Aktiv *)
ELSE
	T_ExchgParam.T_Station1.wState:=T_ExchgParam.T_Station1.wState AND 16#FD;
END_IF;
IF TStation_Work_St1.TControl.xError THEN
	T_ExchgParam.T_Station1.wState:=T_ExchgParam.T_Station1.wState OR 16#4;		(* Stationsfehler Aktiv *)
ELSE
	T_ExchgParam.T_Station1.wState:=T_ExchgParam.T_Station1.wState AND 16#FB;
END_IF;

ptrActivStation:=ADR(TStation_Work_St1);
T_ExchgParam.T_StationCommon.wState:=T_ExchgParam.T_Station1.wState;
END_ACTION
ACTION ProfileManagement:
(* Pointer Profile List Up/Down *)
	RisingEdgePtrProfileListUpDown(CLK:=	T_ExchgParam.T_ProfileCommon.T_ProfileManage.xListProfileUp
										OR T_ExchgParam.T_ProfileCommon.T_ProfileManage.xListProfileDown);
	IF RisingEdgePtrProfileListUpDown.Q THEN
		IF T_ExchgParam.T_ProfileCommon.T_ProfileManage.xListProfileUp THEN
			T_TempActiveState.iPtrListProfile:=T_TempActiveState.iPtrListProfile-5;
			ELSE T_TempActiveState.iPtrListProfile:=T_TempActiveState.iPtrListProfile+5; END_IF
		(* min/max=1/6 *)
		IF T_TempActiveState.iPtrListProfile>(csiMaxProfile - 5) THEN T_TempActiveState.iPtrListProfile:=(csiMaxProfile - 4); END_IF
		IF T_TempActiveState.iPtrListProfile<0 THEN T_TempActiveState.iPtrListProfile:=1; END_IF
		T_ExchgParam.T_ProfileCommon.T_ProfileManage.xListProfileUp:=FALSE;
		T_ExchgParam.T_ProfileCommon.T_ProfileManage.xListProfileDown:=FALSE;
		(* Update display  list *)
		xUpdateProfileList:=TRUE;
	END_IF

(* Update profile list *)
	IF xUpdateProfileList THEN
		xTmp:= 	T_TempActiveState.iPtrListProfile > 0
				AND (T_TempActiveState.iPtrListProfile+4) <= csiMaxProfile;
		IF xTmp THEN
			jj:=1;
			FOR ii:=T_TempActiveState.iPtrListProfile TO T_TempActiveState.iPtrListProfile+4 DO
				T_ExchgParam.T_ProfileCommon.T_ProfileList[jj].iNumber:=ii;
				T_ExchgParam.T_ProfileCommon.T_ProfileList[jj].sName:=T_Profile.T_IDProfileStation[ii].sName;
				jj:=jj+1;
			END_FOR
		END_IF
		(* confirm update *)
		xUpdateProfileList:=FALSE;
		FOR ii:=1 TO 100 DO
			IF (T_Profile.T_IDProfileStation[ii].sName = '') THEN
				T_NovRam.T_Parameter.arZ1AxisCalcEndPosSaveProfile[1,ii]:=0;		(* Wenn kein Profil gespeichert ist, dann kann das zugehörige Inkrementzähler gelöscht werden *)
				T_NovRam.T_Parameter.arZ1CentringCalcEndPosSaveProfile[1,ii]:=0;	(* Wenn kein Profil gespeichert ist, dann kann das zugehörige Inkrementzähler gelöscht werden *)
			END_IF;
		END_FOR;
	END_IF

(* monitor change actual profile common *)
	IF (T_Visu.T_PlcParam.dwActualPage = gT_PageNumber.iHandMode_ProfileMngmt1) OR (T_Visu.T_PlcParam.dwActualPage = gT_PageNumber.iAutoMode_Profile) THEN
		IF T_ExchgParam.T_ProfileCommon.T_Id.iNumber<>iActualActiveProfile THEN
			IF T_Visu.T_CtrleAction.xDone THEN
				(* set value from selected profile *)
				(* save value *)
				T_TempActiveState.iActiveProfile:=T_ExchgParam.T_ProfileCommon.T_Id.iNumber;
				T_ExchgParam.T_ProfileCommon.T_Id.sName
					:=T_Profile.T_IDProfileStation[T_ExchgParam.T_ProfileCommon.T_Id.iNumber].sName;
				iActualActiveProfile:=T_ExchgParam.T_ProfileCommon.T_Id.iNumber;
			END_IF
		END_IF
	END_IF

(* Compare Profile and Process value *)
	T_Profile.T_ProcProfileParameter.T_ProzessData:=T_NovRam.T_Parameter.T_StationWork[gciStationSt1].T_StProcess;
	T_Profile.T_ProcProfileParameter.T_ProfileOnlineChange:=T_NovRam.T_Parameter.T_StationWork[gciStationSt1].T_OnlineChange;

	fbCompareProfileProcessValue(	T_LoadProfileParameter:=T_Profile.T_LoadProfileParameter,
									T_ProfileParameter:=T_Profile.T_ProcProfileParameter);
	T_ExchgParam.T_StationCommon.T_Param_StationWork.T_InfoProcess.xOnlineValueModified:=fbCompareProfileProcessValue.xProcessValueModified;


	T_Profile.T_ProcProfileParameter.T_ProzessData:=T_NovRam.T_Parameter.T_StationWork[gciStationSt1].T_StProcess;
	T_Profile.T_ProcProfileParameter.T_ProfileOnlineChange:=T_NovRam.T_Parameter.T_StationWork[gciStationSt1].T_OnlineChange;

	fbCompareProfileProcessValue(	T_LoadProfileParameter:=T_Profile.T_LoadProfileParameter,
									T_ProfileParameter:=T_Profile.T_ProcProfileParameter);

